(* CODESYS project TcMotion_Axis_v1.0.0.3.library
   DefaultNamespace: Tc3_Motion
   Description: Component Motion OOP Axis
   Author: victorduranm@hotmail.com
   DocFormat: reStructuredText
   Title: TcMotion_Component
   Version: 1.0.0.3
   Company: TcMotion
   Placeholder: TcMotion_Component

Project tree, tasks and I/O mapping:
  libraries: CoDeSys Library Template Interfaces, * (3S - Smart Software Solutions GmbH); Tc2_MC2, * (Beckhoff Automation GmbH); Tc2_MC2_Camming, * (Beckhoff Automation GmbH); Tc2_MC2_FlyingSaw, * (Beckhoff Automation GmbH); Tc2_Standard, * (Beckhoff Automation GmbH); Tc2_System, * (Beckhoff Automation GmbH); Tc3_DriveMotionControl, * (Beckhoff Automation GmbH); Tc3_Module, * (Beckhoff Automation GmbH)
  Component_Axis/
    function block FB_TcAxis_Codesys [ST]: AccelerationProfile, ActualPosition, ActualTorque, ActualVelocity, AxisWarning, CamIn, CombineAxes, CommunicationReady, Direction, ErrorId, GearIn, GearInPos, Halt, HaltSuperimposed, Home, HomeAbsSwitch, IsHomed, LimitSwitchNegative, LimitSwitchPositive, MotionStatus, MoveAbsolute, MoveAdditive, MoveContinuousAbsolute, MoveContinuousRelative, MoveRelative, MoveSuperimposed, MoveVelocity, PhasingAbsolute, PhasingRelative, PositionProfile, Power, PowerOn, ReadBoolParameter, ReadParameter, ReadyForPowerOn, Release, Reset, SetOverride, SetPosition, Simulation, Status, Stop, TorqueControl, VelocityProfile, WriteBoolParameter, WriteParameter
  Examples/
    program CamGearExample [ST]
    program LabelingExample [ST]
    program MAIN_Examples [ST]
    program WareHousingExample [ST]
  MsTestUnit/
    function block FB_Sum [ST]: Sum
  Project Information/
    function F_GetCompany [ST]
    function F_GetTitle [ST]
    function F_GetVersion [ST]
  TwinCAT Library Template/
    Part1Definition/
      Enums/
        data type AXIS_DIRECTION
        data type AXIS_STATUS
        data type E_AxisParameters
        data type MC_BUFFER_MODE
        data type MC_COMBINE_MODE
        data type MC_Direction
        data type MC_Error
        data type MC_ErrorID_Udint
        data type MC_ExecutionMode
        data type MC_Source
        data type MC_StartMode
        data type MC_SYNC_MODE
        data type MOTION_STATUS
      GlobalConstants/
        global variables Constants
      Interfaces/
        interface itfAxis: ActualPosition, ActualTorque, ActualVelocity, Power, ReadBoolParameter, ReadParameter, Release, Reset, SetOverride, SetPosition, WriteBoolParameter, WriteParameter, CombineAxes, GearIn, PhasingAbsolute, PhasingRelative, AccelerationProfile, Halt, HaltSuperimposed, Home, Jog, MoveAbsolute, MoveAdditive, MoveContinuousAbsolute, MoveContinuousRelative, MoveRelative, MoveSuperimposed, MoveVelocity, PositionProfile, Stop, TorqueControl, VelocityProfile, AxisWarning, CommunicationReady, Direction, Error, ErrorId, ErrorId_Udint_Status, Geared, HomeAbsSwitch, IsHomed, LimitSwitchNegative, LimitSwitchPositive, MotionStatus, PowerOn, ReadyForPowerOn, Simulation, Status
        interface itfAxis_Tc2_MC2_Camming: CamIn
        interface itfAxis_Tc2_MC2_FlyingSaw: GearInPos
        interface itfAxisCommand: update
        interface itfCamTable: Select
        interface itfCommand: Abort, Active, Busy, Command, CommandAborted, Done, Error, ErrorId, ErrorID_Udint, Wait
        interface itfContinuousAxisCommand: InVelocity
        interface itfSynchronizedAxisCommand: InSync
      Structs/
        data type MC_CAM_REF
        data type MC_COMMAND_REF
        data type ST_Command
        data type ST_MC
    VendorImplementation/
      function block TcAxis_DMC_Tc3_Direct_Motion_Control [ST]
      function block TcAxis_Tc2_MC2 [ST]: ActualPosition, ActualTorque, ActualVelocity, Power, ReadBoolParameter, ReadParameter, Release, Reset, SetOverride, SetPosition, WriteBoolParameter, WriteParameter, CombineAxes, GearIn, PhasingAbsolute, PhasingRelative, AccelerationProfile, Halt, HaltSuperimposed, Home, Jog, MoveAbsolute, MoveAdditive, MoveContinuousAbsolute, MoveContinuousRelative, MoveRelative, MoveSuperimposed, MoveVelocity, PositionProfile, Stop, TorqueControl, VelocityProfile, AxisWarning, CommunicationReady, Direction, Error, ErrorId, ErrorId_Udint_Status, Geared, HomeAbsSwitch, IsHomed, LimitSwitchNegative, LimitSwitchPositive, MotionStatus, PowerOn, ReadyForPowerOn, Simulation, Status, ACT_Cyclic_Update
      function block TcAxis_Tc2_MC2_Camming [ST]: CamIn
      function block TcAxis_Tc2_MC2_FlyingSaw [ST]: GearInPos
      function block TcAxisCommand [ST]: Abort, Active, Busy, Command, CommandAborted, Done, Error, ErrorId, ErrorID_Udint, Update, Wait
      function block TcCamTable [ST]: Select
      function block TcCommand [ST]: Abort, Active, Busy, Command, CommandAborted, Done, Error, ErrorId, ErrorID_Udint, Wait
      function block TcContinuousAxisCommand [ST]: Abort, Active, Busy, Command, CommandAborted, Done, Error, ErrorId, InVelocity, Update, Wait
      function block TcSynchronizedAxisCommand [ST]: Abort, Active, Busy, Command, CommandAborted, Done, Error, ErrorId, InSync, Update, Wait
  Version/
    global variables Global_Version
  VISUs/
*)

// TwinCAT Library Template/Part1Definition/Enums/AXIS_DIRECTION
{attribute 'qualified_only'}
{attribute 'strict'}
TYPE AXIS_DIRECTION :
(
	DirectionPositive := 0,
	DirectionNegative := 1
);
END_TYPE

// TwinCAT Library Template/Part1Definition/Enums/AXIS_STATUS
{attribute 'qualified_only'}
{attribute 'strict'}
TYPE AXIS_STATUS :
(
	ErrorStop := 0,
	Disabled := 1,
	Stopping := 2,
	Homing := 3,
	Standstill := 4,
	DiscreteMotion := 5,
	ContinuousMotion := 6,
	SynchronizedMotion := 7
);
END_TYPE

// TwinCAT Library Template/Part1Definition/Enums/E_AxisParameters
{attribute 'qualified_only'}
{attribute 'strict'}
TYPE E_AxisParameters :
(
//PLCopen specific parameters Index-Group 0x4000 + ID
    CommandedPosition := 1, //lreal taken from NcToPlc
    SWLimitForward := 2, //lreal IndexOffset= 16#0001_000E
    SWLimitBackward := 3, //lreal IndexOffset= 16#0001_000D
    EnableLimitForward := 4, //bool IndexOffset= 16#0001_000C
    EnableLimitBackward := 5, //bool IndexOffset= 16#0001_000B
    EnablePositionLagMonitoring := 6, //bool IndexOffset= 16#0002_0010
    MaxPositionLag := 7, //lreal IndexOffset= 16#0002_0012
    AxisMaxVelocity := 8, //lreal IndexOffset= 16#0000_0027
    ActualVelocity := 10, //lreal taken from NcToPlc
    CommandedVelocity := 11, //lreal taken from NcToPlc
    AxisDefaultAcceleration := 12, //lreal IndexOffset= 16#0000_0101
    AxisDefaultDeceleration := 14, //lreal IndexOffset= 16#0000_0102
    AxisDefaultJerk := 16, //lreal IndexOffset= 16#0000_0103

//Beckhoff specific parameters Index-Group 0x4000 + ID
    AxisId := 1000, //lreal IndexOffset= 16#0000_0001
    AxisManualVelocitySlow := 1001, //lreal IndexOffset= 16#0000_0008
    AxisManualVelocityFast := 1002, //lreal IndexOffset= 16#0000_0009
    AxisAccMax := 1004, //lreal IndexOffset= 16#0000_0101
    AxisDecMax := 1005, //lreal IndexOffset= 16#0000_0102
    AxisRapidTraverseVelocity := 1009, //lreal IndexOffset= 16#0000_000A
    AxisVelocityToCam := 1012, //lreal IndexOffset= 16#0000_0006
    AxisVelocityFromCam := 1013, //lreal IndexOffset= 16#0000_0007
    AxisJogIncrementForward := 1014, //lreal IndexOffset= 16#0000_0018
    AxisJogIncrementBackward := 1015, //lreal IndexOffset= 16#0000_0019
    MaxPositionLagFilterTime := 1022, //lreal IndexOffset= 16#0002_0013
    AxisEnPositionRangeMonitoring := 1023, //bool IndexOffset= 16#0000_000F
    AxisPositionRangeWindow := 1024, //lreal IndexOffset= 16#0000_0010
    AxisEnTargetPositionMonitoring:= 1025, //bool IndexOffset= 16#0000_0015
    AxisTargetPositionWindow := 1026, //lreal IndexOffset= 16#0000_0016
    AxisTargetPositionMonitoringTime := 1027, //lreal IndexOffset= 16#0000_0017
    AxisEnInTargetTimeout := 1028, //bool IndexOffset= 16#0000_0029
    AxisInTargetTimeout := 1029, //lreal IndexOffset= 16#0000_002A
    AxisEnMotionMonitoring := 1030, //bool IndexOffset= 16#0000_0011
    AxisMotionMonitoringWindow := 1031, //lreal IndexOffset= 16#0000_0028
    AxisMotionMonitoringTime := 1032, //lreal IndexOffset= 16#0000_0012
    AxisDelayTimeVeloPosition := 1033, //lreal IndexOffset= 16#0000_0104
    AxisEnLoopingDistance := 1034, //bool IndexOffset= 16#0000_0013
    AxisLoopingDistance := 1035, //lreal IndexOffset= 16#0000_0014
    AxisEnBacklashCompensation := 1036, //bool IndexOffset= 16#0000_002B
    AxisBacklash := 1037, //lreal IndexOffset= 16#0000_002C
    AxisEnDataPersistence := 1038, //bool IndexOffset= 16#0000_0030
    AxisRefVeloOnRefOutput := 1039, //lreal IndexOffset= 16#0003_0101
    AxisOverrideType := 1040, //lreal IndexOffset= 16#0000_0105
    //new since 4/2007
    AxisEncoderOffset := 1042, //lreal IndexOffset= 16#0001_0007
    AxisEncoderDirectionInverse := 1043, //bool IndexOffset= 16#0001_0008
    AxisEncoderMask := 1044, //dword IndexOffset= 16#0001_0015
    AxisEncoderModuloValue := 1045, //lreal IndexOffset= 16#0001_0009
    AxisModuloToleranceWindow := 1046, //lreal IndexOffset= 16#0001_001B
    AxisEnablePosCorrection := 1047, //bool IndexOffset= 16#0001_0016
    AxisPosCorrectionFilterTime := 1048, //lreal IndexOffset= 16#0001_0017
    //new since 1/2010
    AxisUnitInterpretation := 1049, //lreal IndexOffset= 16#0000_0026
    AxisMotorDirectionInverse := 1050, //bool  IndexOffset= 16#0003_0006
    //new since 1/2011
    AxisCycleTime := 1051, //lreal IndexOffset= 16#0000_0004
    //new since 5/2011
    AxisFastStopSignalType := 1052, //dword IndexOffset= 16#0000_001E
    AxisFastAcc := 1053, //lreal IndexOffset= 16#0000_010A
    AxisFastDec := 1054, //lreal IndexOffset= 16#0000_010B
    AxisFastJerk := 1055, //lreal IndexOffset= 16#0000_010C
    // new since 1/2012 *)
    AxisEncoderScalingNumerator := 1056, //lreal IndexOffset= 16#0001_0023 - available in Tc3
    AxisEncoderScalingDenominator := 1057, //lreal IndexOffset= 16#0001_0024 - available in Tc3
    (* new since 7/2016 *)
    AxisVeloJumpFactor := 1060, //lreal IndexOffset= 16#0000_0106
    AxisToleranceBallAuxAxis := 1061, //lreal IndexOffset= 16#0000_0108
    AxisMaxPositionDeviationAuxAxis := 1062, //lreal IndexOffset= 16#0000_0109
    AxisErrorPropagationMode := 1063, //dword IndexOffset= 16#0000_001A
    AxisErrorPropagationDelay := 1064, //lreal IndexOffset= 16#0000_001B
    AxisCoupleSlaveToActualValues := 1065, //bool IndexOffset= 16#0000_001C
    AxisAllowMotionCmdToSlaveAxis := 1066, //bool IndexOffset= 16#0000_0020
    AxisAllowMotionCmdToExtSetAxis := 1067, //bool IndexOffset= 16#0000_0021
    AxisEncoderSubMask := 1068, //dword IndexOffset= 16#0001_0108
    AxisEncoderReferenceSystem := 1069, //dword IndexOffset= 16#0001_0019
    AxisEncoderPositionFilterPT1 := 1070, //lreal IndexOffset= 16#0001_0010
    AxisEncoderVelocityFilterPT1 := 1071, //lreal IndexOffset= 16#0001_0011
    AxisEncoderAccelerationFilterPT1 := 1072, //lreal IndexOffset= 16#0001_0012
    AxisEncoderMode := 1073, //dword IndexOffset= 16#0001_000A
    AxisEncoderHomingInvDirCamSearch := 1074, //bool IndexOffset= 16#0001_0101
    AxisEncoderHomingInvDirSyncSearch := 1075, //bool IndexOffset= 16#0001_0102
    AxisEncoderHomingCalibValue := 1076, //lreal IndexOffset= 16#0001_0103
    AxisEncoderReferenceMode := 1077, //dword IndexOffset= 16#0001_0107
    AxisRefVeloOutputRatio := 1078, //lreal IndexOffset= 16#0003_0102
    AxisDrivePositionOutputScaling := 1079, //lreal IndexOffset= 16#0003_0109
    AxisDriveVelocityOutputScaling := 1080, //lreal IndexOffset= 16#0003_0105
    AxisDriveVelocityOutputDelay := 1081, //lreal IndexOffset= 16#0003_010D
    AxisDriveMinOutputLimitation := 1082, //lreal IndexOffset= 16#0003_000B
    AxisDriveMaxOutputLimitation := 1083, //lreal IndexOffset= 16#0003_000C
    AxisTorqueInputScaling := 1084, //lreal IndexOffset= 16#0003_0031 - available in Tc3
    AxisTorqueInputFilterPT1 := 1085, //lreal IndexOffset= 16#0003_0032 - available in Tc3
    AxisTorqueDerivationInputFilterPT1 := 1086, //lreal IndexOffset= 16#0003_0033 - available in Tc3
    AxisTorqueOutputScaling := 1087, //lreal IndexOffset= 16#0003_010B
    AxisTorqueOutputDelay := 1088, //lreal IndexOffset= 16#0003_010F
    AxisAccelerationOutputScaling := 1089, //lreal IndexOffset= 16#0003_010A
    AxisAccelerationOutputDelay := 1090, //lreal IndexOffset= 16#0003_010E
    AxisDrivePositionOutputSmoothFilterType := 1091, //dword IndexOffset= 16#0003_0110
    AxisDrivePositionOutputSmoothFilterTime := 1092, //lreal IndexOffset= 16#0003_0111
    AxisDrivePositionOutputSmoothFilterOrder := 1093, //dword IndexOffset= 16#0003_0112
    AxisDriveMode := 1094, //dword IndexOffset= 16#0003_000A
    AxisDriftCompensationOffset := 1095, //lreal IndexOffset= 16#0003_0104
    AxisPositionControlKv := 1096, //lreal IndexOffset= 16#0002_0102
    AxisCtrlVelocityPreCtrlWeight := 1097, //lreal IndexOffset= 16#0002_000B
    AxisControllerMode := 1098, //dword IndexOffset= 16#0002_000A
    AxisCtrlAutoOffset := 1099, //bool IndexOffset= 16#0002_0110
    AxisCtrlAutoOffsetTimer := 1100, //lreal IndexOffset= 16#0002_0115
    AxisCtrlAutoOffsetLimit := 1101, //lreal IndexOffset= 16#0002_0114
    AxisSlaveCouplingControlKcp := 1102, //lreal IndexOffset= 16#0002_010F
    AxisCtrlOutputLimit := 1103, //lreal IndexOffset= 16#0002_0100

//Beckhoff specific axis status information - READ ONLY Index-Group 0x4100 + ID
    AxisTargetPosition := 2000, //lreal IndexOffset= 16#0000_0013
    AxisRemainingTimeToGo := 2001, //lreal IndexOffset= 16#0000_0014
    AxisRemainingDistanceToGo := 2002, //lreal IndexOffset= 16#0000_0022, 16#0000_0042

//Beckhoff specific axis functions
    //read/write gear ratio of a slave
    AxisGearRatio := 3000, //lreal read: IndexGroup=0x4100+ID, IdxOffset=16#0000_0022,
                                 //write:IndexGroup=0x4200+ID, IdxOffset=16#0000_0042

//Beckhoff specific other parameters
    //new since 1/2011
    NcSafCycleTime := 4000, //lreal IndexOffset= 16#0000_0010
    NcSvbCycleTime := 4001 //lreal IndexOffset= 16#0000_0012

);
END_TYPE

// TwinCAT Library Template/Part1Definition/Enums/MC_BUFFER_MODE
{attribute 'qualified_only'}
{attribute 'strict'}
TYPE MC_BUFFER_MODE :
(
	mcAborting := 0,
	mcBuffered := 1,
	mcBlendingLow := 2,
	mcBlendingPrevious := 3,
	mcBlendingNext := 4,
	mcBlendingHigh := 5
);
END_TYPE

// TwinCAT Library Template/Part1Definition/Enums/MC_COMBINE_MODE
{attribute 'qualified_only'}
{attribute 'strict'}
TYPE MC_COMBINE_MODE :
(
	enum_member := 0
);
END_TYPE

// TwinCAT Library Template/Part1Definition/Enums/MC_Direction
{attribute 'qualified_only'}
{attribute 'strict'}
TYPE MC_Direction :
(
	mcPositiveDirection := 0,
	mcShortestWay := 1,
	mcNegativeDirection := 2,
	mcCurrentDirection := 3
);
END_TYPE

// TwinCAT Library Template/Part1Definition/Enums/MC_Error
{attribute 'qualified_only'}
//{attribute 'conditionalshow' := 'SomeText'}
//{attribute 'conditionalshow'}
//{attribute 'hide'}
TYPE MC_Error : (NO_ERROR, TIME_OUT); END_TYPE

// TwinCAT Library Template/Part1Definition/Enums/MC_ErrorID_Udint
TYPE MC_ErrorID_Udint : UDINT; END_TYPE

// TwinCAT Library Template/Part1Definition/Enums/MC_ExecutionMode
{attribute 'qualified_only'}
{attribute 'strict'}
TYPE MC_ExecutionMode :
(
	mcImmediatly := 0,
	mcQueue := 1
);
END_TYPE

// TwinCAT Library Template/Part1Definition/Enums/MC_Source
{attribute 'qualified_only'}
{attribute 'strict'}
TYPE MC_Source :
(
	mcSetValue := 0,
	mcActualValue := 1
);
END_TYPE

// TwinCAT Library Template/Part1Definition/Enums/MC_StartMode
{attribute 'qualified_only'}
{attribute 'strict'}
TYPE MC_StartMode :
(
	mcAbsolute := 0,
	mcRelative := 1,
	mcRampIn := 2
);
END_TYPE

// TwinCAT Library Template/Part1Definition/Enums/MC_SYNC_MODE
{attribute 'qualified_only'}
{attribute 'strict'}
TYPE MC_SYNC_MODE :
(
	enum_member := 0
);
END_TYPE

// TwinCAT Library Template/Part1Definition/Enums/MOTION_STATUS
{attribute 'qualified_only'}
{attribute 'strict'}
TYPE MOTION_STATUS :
(
	ConstantVelocity := 0,
	Accelerating := 1,
	Decelerating :=2
);
END_TYPE

// TwinCAT Library Template/Part1Definition/Structs/MC_CAM_REF
TYPE MC_CAM_REF :
STRUCT
END_STRUCT
END_TYPE

// TwinCAT Library Template/Part1Definition/Structs/MC_COMMAND_REF
TYPE MC_COMMAND_REF :
STRUCT
	CommandId: INT;
END_STRUCT
END_TYPE

// TwinCAT Library Template/Part1Definition/Structs/ST_Command
TYPE ST_Command :
STRUCT
	Active 			: BOOL;
	Busy 			: BOOL;
	Command 		: MC_COMMAND_REF;
	CommandAborted 	: BOOL;
	Done           	: BOOL;
	Error    		: BOOL;
	ErrorId        	: MC_Error;
	ErrorID_Udint	: MC_ErrorID_Udint;
END_STRUCT
END_TYPE

// TwinCAT Library Template/Part1Definition/Structs/ST_MC
TYPE ST_MC :
STRUCT
	Power 			: Tc2_MC2.MC_POWER;
	MoveAbsolute 	: Tc2_MC2.MC_MoveAbsolute;	
	MoveRelative 	: Tc2_MC2.MC_MoveRelative;
END_STRUCT
END_TYPE

// TwinCAT Library Template/Part1Definition/GlobalConstants/Constants
//{attribute 'conditionalshow' := 'SomeText'}
//{attribute 'conditionalshow'}
//{attribute 'hide'}
VAR_GLOBAL CONSTANT
END_VAR

// Version/Global_Version
{attribute 'TcGenerated'}
{attribute 'no-analysis'}
{attribute 'linkalways'}
// This function has been automatically generated from the project information.
VAR_GLOBAL CONSTANT
	{attribute 'const_non_replaced'}
	stLibVersion_TcMotion_Component : ST_LibVersion := (iMajor := 1, iMinor := 0, iBuild := 0, iRevision := 3, nFlags := 0, sVersion := '1.0.0.3');
END_VAR

// Component_Axis/FB_TcAxis_Codesys
FUNCTION_BLOCK FB_TcAxis_Codesys IMPLEMENTS TMP.itfAxis
VAR_INPUT
END_VAR
VAR_OUTPUT
END_VAR
VAR
END_VAR

{warning 'Agregar implementación de método'}
METHOD AccelerationProfile : itfCommand
VAR_INPUT
	TimeScale	: REAL;
	AccelerationScale	: REAL;
	Offset	: REAL;
	BufferMode	: MC_BUFFER_MODE;
END_VAR
// NETWORK 1
END_METHOD

{warning 'Agregar implementación de propiedad'}
PROPERTY ActualPosition : REAL
GET
// NETWORK 1
END_GET
END_PROPERTY

{warning 'Agregar implementación de propiedad'}
PROPERTY ActualTorque : REAL
GET
// NETWORK 1
END_GET
END_PROPERTY

{warning 'Agregar implementación de propiedad'}
PROPERTY ActualVelocity : REAL
GET
// NETWORK 1
END_GET
END_PROPERTY

{warning 'Agregar implementación de propiedad'}
PROPERTY AxisWarning : BOOL
GET
// NETWORK 1
END_GET
END_PROPERTY

{warning 'Agregar implementación de método'}
METHOD CamIn : itfSynchronizedAxisCommand
VAR_INPUT
	Master	: itfAxis;
	MasterOffset	: REAL;
	SlaveOffset	: REAL;
	MasterScaling	: REAL;
	SlaveScaling	: REAL;
	MasterStartDistance	: REAL;
	MasterSyncPosition	: REAL;
	StartMode	: MC_StartMode;
	MasterValueSource	: MC_Source;
	CamTable	: itfCamTable;
	BufferMode	: MC_BUFFER_MODE;
END_VAR
// NETWORK 1
END_METHOD

{warning 'Agregar implementación de método'}
METHOD CombineAxes : itfSynchronizedAxisCommand
VAR_INPUT
	Master1	: itfAxis;
	Master2	: itfAxis;
	CombineMode	: MC_COMBINE_MODE;
	GearRatioNumeratorM1	: INT;
	GearRatioDenominatorM1	: INT;
	GearRatioNumeratorM2	: INT;
	GearRatioDenominatorM2	: INT;
	MasterValueSourceM1	: MC_SOURCE;
	MasterValueSourceM2	: MC_SOURCE;
	BufferMode	: MC_BUFFER_MODE;
END_VAR
// NETWORK 1
END_METHOD

{warning 'Agregar implementación de propiedad'}
PROPERTY CommunicationReady : BOOL
GET
// NETWORK 1
END_GET
END_PROPERTY

{warning 'Agregar implementación de propiedad'}
PROPERTY Direction : AXIS_DIRECTION
GET
// NETWORK 1
END_GET
END_PROPERTY

{warning 'Agregar implementación de propiedad'}
PROPERTY ErrorId : WORD
GET
// NETWORK 1
END_GET
END_PROPERTY

{warning 'Agregar implementación de método'}
METHOD GearIn : itfSynchronizedAxisCommand
VAR_INPUT
	Master	: itfAxis;
	Ratio	: REAL;
	MasterValueSource	: INT;
	Acceleration	: REAL;
	Deceleration	: REAL;
	Jerk	: REAL;
	BufferMode	: MC_BUFFER_MODE;
END_VAR
// NETWORK 1
END_METHOD

{warning 'Agregar implementación de método'}
METHOD GearInPos : itfSynchronizedAxisCommand
VAR_INPUT
	Master	: itfAxis;
	RatioNumerator	: REAL;
	RatioDenominator	: REAL;
	MasterValueSource	: MC_SOURCE;
	MasterSyncPosition	: REAL;
	SlaveSyncPosition	: REAL;
	SyncMode	: MC_SYNC_MODE;
	MasterStartDistance	: REAL;
	Velocity	: REAL;
	Acceleration	: REAL;
	Deceleration	: REAL;
	Jerk	: REAL;
	BufferMode	: MC_BUFFER_MODE;
END_VAR
// NETWORK 1
END_METHOD

{warning 'Agregar implementación de método'}
METHOD Halt : itfAxisCommand
VAR_INPUT
	Deceleration	: REAL;
	Jerk	: REAL;
	BufferMode	: MC_BUFFER_MODE;
END_VAR
// NETWORK 1
END_METHOD

{warning 'Agregar implementación de método'}
METHOD HaltSuperimposed : itfAxisCommand
VAR_INPUT
	Deceleration	: REAL;
	Jerk	: REAL;
END_VAR
// NETWORK 1
END_METHOD

{warning 'Agregar implementación de método'}
METHOD Home : itfAxisCommand
VAR_INPUT
	Position	: REAL;
	Velocity	: REAL;
	EndVelocity	: REAL;
	Acceleration	: REAL;
	Deceleration	: REAL;
	Jerk	: REAL;
	Direction	: MC_Direction;
	HomingMode	: INT;
	BufferMode	: MC_BUFFER_MODE;
END_VAR
// NETWORK 1
END_METHOD

{warning 'Agregar implementación de propiedad'}
PROPERTY HomeAbsSwitch : BOOL
GET
// NETWORK 1
END_GET
END_PROPERTY

{warning 'Agregar implementación de propiedad'}
PROPERTY IsHomed : BOOL
GET
// NETWORK 1
END_GET
END_PROPERTY

{warning 'Agregar implementación de propiedad'}
PROPERTY LimitSwitchNegative : BOOL
GET
// NETWORK 1
END_GET
END_PROPERTY

{warning 'Agregar implementación de propiedad'}
PROPERTY LimitSwitchPositive : BOOL
GET
// NETWORK 1
END_GET
END_PROPERTY

{warning 'Agregar implementación de propiedad'}
PROPERTY MotionStatus : MOTION_STATUS
GET
// NETWORK 1
END_GET
END_PROPERTY

{warning 'Agregar implementación de método'}
METHOD MoveAbsolute : itfAxisCommand
VAR_INPUT
	Position	: REAL;
	Velocity	: REAL;
	Acceleration	: REAL;
	Deceleration	: REAL;
	Jerk	: REAL;
	Direction	: MC_Direction;
	BufferMode	: MC_BUFFER_MODE;
END_VAR
// NETWORK 1
END_METHOD

{warning 'Agregar implementación de método'}
METHOD MoveAdditive : itfAxisCommand
VAR_INPUT
	Distance	: REAL;
	Velocity	: REAL;
	Acceleration	: REAL;
	Deceleration	: REAL;
	Jerk	: REAL;
	BufferMode	: MC_BUFFER_MODE;
END_VAR
// NETWORK 1
END_METHOD

{warning 'Agregar implementación de método'}
METHOD MoveContinuousAbsolute : itfContinuousAxisCommand
VAR_INPUT
	Position	: REAL;
	EndVelocity	: REAL;
	Velocity	: REAL;
	Acceleration	: REAL;
	Deceleration	: REAL;
	Jerk	: REAL;
	Direction	: MC_DIRECTION;
	BufferMode	: MC_BUFFER_MODE;
END_VAR
// NETWORK 1
END_METHOD

{warning 'Agregar implementación de método'}
METHOD MoveContinuousRelative : itfContinuousAxisCommand
VAR_INPUT
	Distance	: REAL;
	EndVelocity	: REAL;
	Velocity	: REAL;
	Acceleration	: REAL;
	Deceleration	: REAL;
	Jerk	: REAL;
	Direction	: MC_DIRECTION;
	BufferMode	: MC_BUFFER_MODE;
END_VAR
// NETWORK 1
END_METHOD

{warning 'Agregar implementación de método'}
METHOD MoveRelative : itfAxisCommand
VAR_INPUT
	Distance	: REAL;
	Velocity	: REAL;
	Acceleration	: REAL;
	Deceleration	: REAL;
	Jerk	: REAL;
	BufferMode	: MC_BUFFER_MODE;
END_VAR
// NETWORK 1
END_METHOD

{warning 'Agregar implementación de método'}
METHOD MoveSuperimposed : itfAxisCommand
VAR_INPUT
	Distance	: REAL;
	VelocityDiff	: REAL;
	Acceleration	: REAL;
	Deceleration	: REAL;
	Jerk	: REAL;
END_VAR
// NETWORK 1
END_METHOD

{warning 'Agregar implementación de método'}
METHOD MoveVelocity : itfContinuousAxisCommand
VAR_INPUT
	Velocity	: REAL;
	Acceleration	: REAL;
	Deceleration	: REAL;
	Jerk	: REAL;
	Direction	: MC_Direction;
	BufferMode	: MC_BUFFER_MODE;
END_VAR
// NETWORK 1
END_METHOD

{warning 'Agregar implementación de método'}
METHOD PhasingAbsolute : itfSynchronizedAxisCommand
VAR_INPUT
	Master	: itfAxis;
	PhaseShift	: REAL;
	Velocity	: REAL;
	Acceleration	: REAL;
	Deceleration	: REAL;
	Jerk	: REAL;
	BufferMode	: MC_BUFFER_MODE;
END_VAR
// NETWORK 1
END_METHOD

{warning 'Agregar implementación de método'}
METHOD PhasingRelative : itfSynchronizedAxisCommand
VAR_INPUT
	Master	: itfAxis;
	PhaseShift	: REAL;
	Velocity	: REAL;
	Acceleration	: REAL;
	Deceleration	: REAL;
	Jerk	: REAL;
	BufferMode	: MC_BUFFER_MODE;
END_VAR
// NETWORK 1
END_METHOD

{warning 'Agregar implementación de método'}
METHOD PositionProfile : itfCommand
VAR_INPUT
	TimeScale	: REAL;
	PositionScale	: REAL;
	Offset	: REAL;
	BufferMode	: MC_BUFFER_MODE;
END_VAR
// NETWORK 1
END_METHOD

{warning 'Agregar implementación de método'}
METHOD Power : itfCommand
VAR_INPUT
	Enable	: BOOL;
	EnablePositive	: BOOL;
	EnableNegative	: BOOL;
END_VAR
// NETWORK 1
END_METHOD

{warning 'Agregar implementación de propiedad'}
PROPERTY PowerOn : BOOL
GET
// NETWORK 1
END_GET
END_PROPERTY

{warning 'Agregar implementación de método'}
METHOD ReadBoolParameter : MC_Error
VAR_INPUT
	ParameterNumber	: INT;
END_VAR
VAR_OUTPUT
	Value	: BOOL;
END_VAR
// NETWORK 1
END_METHOD

{warning 'Agregar implementación de método'}
METHOD ReadParameter : MC_Error
VAR_INPUT
	ParameterNumber	: INT;
END_VAR
VAR_OUTPUT
	Value	: REAL;
END_VAR
// NETWORK 1
END_METHOD

{warning 'Agregar implementación de propiedad'}
PROPERTY ReadyForPowerOn : BOOL
GET
// NETWORK 1
END_GET
END_PROPERTY

{warning 'Agregar implementación de método'}
METHOD Release : MC_Error
// NETWORK 1
END_METHOD

{warning 'Agregar implementación de método'}
METHOD Reset : itfCommand
// NETWORK 1
END_METHOD

{warning 'Agregar implementación de método'}
METHOD SetOverride : MC_Error
VAR_INPUT
	VelFactor	: REAL;
	AccFactor	: REAL;
	JerkFactor	: REAL;
END_VAR
// NETWORK 1
END_METHOD

{warning 'Agregar implementación de método'}
METHOD SetPosition : itfCommand
VAR_INPUT
	Position	: REAL;
	Relative	: BOOL;
	ExecutionMode	: MC_ExecutionMode;
END_VAR
// NETWORK 1
END_METHOD

{warning 'Agregar implementación de propiedad'}
PROPERTY Simulation : BOOL
GET
// NETWORK 1
END_GET
END_PROPERTY

{warning 'Agregar implementación de propiedad'}
PROPERTY Status : AXIS_STATUS
GET
// NETWORK 1
END_GET
END_PROPERTY

{warning 'Agregar implementación de método'}
METHOD Stop : itfAxisCommand
VAR_INPUT
	Deceleration	: REAL;
	Jerk	: REAL;
END_VAR
// NETWORK 1
END_METHOD

{warning 'Agregar implementación de método'}
METHOD TorqueControl : itfAxisCommand
VAR_INPUT
	Torque	: REAL;
	TorqueRamp	: REAL;
	Velocity	: REAL;
	Acceleration	: REAL;
	Deceleration	: REAL;
	Jerk	: REAL;
	Direction	: MC_DIRECTION;
	BufferMode	: MC_BUFFER_MODE;
END_VAR
// NETWORK 1
END_METHOD

{warning 'Agregar implementación de método'}
METHOD VelocityProfile : itfCommand
VAR_INPUT
	TimeScale	: REAL;
	VelocityScale	: REAL;
	Offset	: REAL;
	BufferMode	: MC_BUFFER_MODE;
END_VAR
// NETWORK 1
END_METHOD

{warning 'Agregar implementación de método'}
METHOD WriteBoolParameter : MC_Error
VAR_INPUT
	ParameterNumber	: INT;
	Value	: BOOL;
END_VAR
// NETWORK 1
END_METHOD

{warning 'Agregar implementación de método'}
METHOD WriteParameter : MC_Error
VAR_INPUT
	ParameterNumber	: INT;
	Value	: REAL;
END_VAR
// NETWORK 1
END_METHOD

END_FUNCTION_BLOCK

// TwinCAT Library Template/Part1Definition/Interfaces/itfAxis
INTERFACE itfAxis

{warning 'add property implementation'}
PROPERTY ActualPosition : REAL
GET
END_GET
END_PROPERTY

{warning 'add property implementation'}
PROPERTY ActualTorque : REAL
GET
END_GET
END_PROPERTY

{warning 'add property implementation'}
PROPERTY ActualVelocity : REAL
GET
END_GET
END_PROPERTY

{attribute 'TcRpcEnable'}
METHOD Power 		: itfCommand
VAR_INPUT
	Enable			: BOOL;
	EnablePositive	: BOOL;
	EnableNegative	: BOOL;
END_VAR
END_METHOD

{warning 'add method implementation '}
METHOD ReadBoolParameter 	: MC_Error
VAR_INPUT
	ParameterNumber			: INT;
END_VAR
VAR_OUTPUT
	Value					: BOOL;
END_VAR
END_METHOD

{warning 'add method implementation '}
METHOD ReadParameter 	: MC_Error
VAR_INPUT
	ParameterNumber		: INT;
END_VAR
VAR_OUTPUT
	Value				: REAL;
END_VAR
END_METHOD

{warning 'add method implementation '}
METHOD Release : MC_Error
END_METHOD

{attribute 'TcRpcEnable'}
METHOD Reset : itfCommand
END_METHOD

{warning 'add method implementation '}
METHOD SetOverride 	: MC_Error
VAR_INPUT
	VelFactor		: REAL;
	AccFactor		: REAL;
	JerkFactor		: REAL;
END_VAR
END_METHOD

{warning 'add method implementation '}
METHOD SetPosition 	: itfCommand
VAR_INPUT
	Position		: REAL;
	Relative		: BOOL;
//	ExecutionMode	: MC_ExecutionMode;
	ExecutionMode	: Tc2_MC2.ST_SetPositionOptions;
END_VAR
END_METHOD

{warning 'add method implementation '}
METHOD WriteBoolParameter 	: MC_Error
VAR_INPUT
	ParameterNumber			: INT;
	Value					: BOOL;
END_VAR
END_METHOD

{warning 'add method implementation '}
METHOD WriteParameter 	: MC_Error
VAR_INPUT
	ParameterNumber		: INT;
	Value				: REAL;
END_VAR
END_METHOD

{warning 'add method implementation '}
METHOD CombineAxes 			: itfSynchronizedAxisCommand
VAR_INPUT
	Master1					: itfAxis;
	Master2					: itfAxis;
	CombineMode				: MC_COMBINE_MODE;
	GearRatioNumeratorM1	: INT;
	GearRatioDenominatorM1	: INT;
	GearRatioNumeratorM2	: INT;
	GearRatioDenominatorM2	: INT;
	MasterValueSourceM1		: MC_SOURCE;
	MasterValueSourceM2		: MC_SOURCE;
	BufferMode				: MC_BUFFER_MODE;
END_VAR
END_METHOD

{attribute 'TcRpcEnable'}
METHOD GearIn 			: itfSynchronizedAxisCommand
VAR_INPUT
//	Master				: itfAxis;
//	Master				: Tc2_MC2.AXIS_REF;
//	Slave				: Tc2_MC2.AXIS_REF;		
//	Ratio				: REAL;
//	MasterValueSource	: INT;
	RatioNumerator		: LREAL;
	RatioDenominator	: UINT;
	Acceleration		: REAL;
	Deceleration		: REAL;
	Jerk				: REAL;
	BufferMode			: MC_BUFFER_MODE;
//	BufferMode			: Tc2_MC2.MC_BufferMode;
//	Options             : Tc2_MC2.ST_GearInOptions;
END_VAR

VAR_IN_OUT 
	Slave				: Tc2_MC2.AXIS_REF;	
END_VAR
END_METHOD

{warning 'add method implementation '}
METHOD PhasingAbsolute 	: itfSynchronizedAxisCommand
VAR_INPUT
//	Master				: itfAxis;
	Master				: Tc2_MC2.AXIS_REF;
	Slave				: Tc2_MC2.AXIS_REF;		
	PhaseShift			: REAL;
	Velocity			: REAL;
	Acceleration		: REAL;
	Deceleration		: REAL;
	Jerk				: REAL;
	BufferMode			: MC_BUFFER_MODE;
END_VAR
END_METHOD

{warning 'add method implementation '}
METHOD PhasingRelative 	: itfSynchronizedAxisCommand
VAR_INPUT
//	Master				: itfAxis;
	Master				: Tc2_MC2.AXIS_REF;
	Slave				: Tc2_MC2.AXIS_REF;		
	PhaseShift			: REAL;
	Velocity			: REAL;
	Acceleration		: REAL;
	Deceleration		: REAL;
	Jerk				: REAL;
	BufferMode			: MC_BUFFER_MODE;
END_VAR
END_METHOD

{warning 'add method implementation '}
METHOD AccelerationProfile 	: itfCommand
VAR_INPUT
	TimeScale				: REAL;
	AccelerationScale		: REAL;
	Offset					: REAL;
	BufferMode				: MC_BUFFER_MODE;
END_VAR
END_METHOD

{warning 'add method implementation '}
METHOD Halt 		: itfAxisCommand
VAR_INPUT
	Deceleration	: REAL;
	Jerk			: REAL;
	BufferMode		: MC_BUFFER_MODE;
END_VAR
END_METHOD

{warning 'add method implementation '}
METHOD HaltSuperimposed : itfAxisCommand
VAR_INPUT
	Deceleration		: REAL;
	Jerk				: REAL;
END_VAR
END_METHOD

{warning 'add method implementation '}
METHOD Home 		: itfAxisCommand
VAR_INPUT
	Position		: REAL;
	Velocity		: REAL;
	EndVelocity		: REAL;
	Acceleration	: REAL;
	Deceleration	: REAL;
	Jerk			: REAL;
	Direction		: MC_Direction;
	HomingMode		: INT;
	BufferMode		: MC_BUFFER_MODE;
END_VAR
END_METHOD

{warning 'add method implementation '}
METHOD Jog 			: itfAxisCommand
VAR_INPUT
    JogForward 		: BOOL;
    JogBackwards 	: BOOL;
    Mode     		: Tc2_MC2.E_JogMode;
    Position        : LREAL;
    Velocity        : LREAL;
    Acceleration 	: LREAL;
    Deceleration 	: LREAL;
    Jerk     		: LREAL;
END_VAR
END_METHOD

{attribute 'TcRpcEnable'}
METHOD MoveAbsolute : itfAxisCommand
VAR_INPUT
	Position		: REAL;
	Velocity		: REAL;
	Acceleration	: REAL;
	Deceleration	: REAL;
	Jerk			: REAL;
	Direction		: MC_Direction;
	BufferMode		: MC_BUFFER_MODE;
END_VAR
END_METHOD

{warning 'add method implementation '}
METHOD MoveAdditive : itfAxisCommand
VAR_INPUT
	Distance		: REAL;
	Velocity		: REAL;
	Acceleration	: REAL;
	Deceleration	: REAL;
	Jerk			: REAL;
	BufferMode		: MC_BUFFER_MODE;
END_VAR
END_METHOD

{warning 'add method implementation '}
METHOD MoveContinuousAbsolute 	: itfContinuousAxisCommand
VAR_INPUT
	Position					: REAL;
	EndVelocity					: REAL;
	Velocity					: REAL;
	Acceleration				: REAL;
	Deceleration				: REAL;
	Jerk						: REAL;
	Direction					: MC_DIRECTION;
	BufferMode					: MC_BUFFER_MODE;
END_VAR
END_METHOD

{warning 'add method implementation '}
METHOD MoveContinuousRelative 	: itfContinuousAxisCommand
VAR_INPUT
	Distance					: REAL;
	EndVelocity					: REAL;
	Velocity					: REAL;
	Acceleration				: REAL;
	Deceleration				: REAL;
	Jerk						: REAL;
	Direction					: MC_DIRECTION;
	BufferMode					: MC_BUFFER_MODE;
END_VAR
END_METHOD

{attribute 'TcRpcEnable'}
METHOD MoveRelative : itfAxisCommand
VAR_INPUT
	Distance		: REAL;
	Velocity		: REAL;
	Acceleration	: REAL;
	Deceleration	: REAL;
	Jerk			: REAL;
	BufferMode		: MC_BUFFER_MODE;
END_VAR
END_METHOD

{warning 'add method implementation '}
METHOD MoveSuperimposed : itfAxisCommand
VAR_INPUT
	Distance			: REAL;
	VelocityDiff		: REAL;
	Acceleration		: REAL;
	Deceleration		: REAL;
	Jerk				: REAL;
END_VAR
END_METHOD

{warning 'add method implementation '}
METHOD MoveVelocity : itfContinuousAxisCommand
VAR_INPUT
	Velocity		: REAL;
	Acceleration	: REAL;
	Deceleration	: REAL;
	Jerk			: REAL;
	Direction		: MC_Direction;
	BufferMode		: MC_BUFFER_MODE;
END_VAR
END_METHOD

{warning 'add method implementation '}
METHOD PositionProfile : itfCommand
VAR_INPUT
	TimeScale			: REAL;
	PositionScale		: REAL;
	Offset				: REAL;
	BufferMode			: MC_BUFFER_MODE;
END_VAR
END_METHOD

{warning 'add method implementation '}
METHOD Stop 		: itfAxisCommand
VAR_INPUT
	Deceleration	: REAL;
	Jerk			: REAL;
END_VAR
END_METHOD

{warning 'add method implementation '}
METHOD TorqueControl	: itfAxisCommand
VAR_INPUT
	Torque				: REAL;
	TorqueRamp			: REAL;
	Velocity			: REAL;
	Acceleration		: REAL;
	Deceleration		: REAL;
	Jerk				: REAL;
	Direction			: MC_DIRECTION;
	BufferMode			: MC_BUFFER_MODE;
END_VAR
END_METHOD

{warning 'add method implementation '}
METHOD VelocityProfile 	: itfCommand
VAR_INPUT
	TimeScale			: REAL;
	VelocityScale		: REAL;
	Offset				: REAL;
	BufferMode			: MC_BUFFER_MODE;
END_VAR
END_METHOD

{warning 'add property implementation'}
PROPERTY AxisWarning : BOOL
GET
END_GET
END_PROPERTY

{warning 'add property implementation'}
PROPERTY CommunicationReady : BOOL
GET
END_GET
END_PROPERTY

{warning 'add property implementation'}
PROPERTY Direction : AXIS_DIRECTION
GET
END_GET
END_PROPERTY

PROPERTY Error : BOOL
GET
END_GET
END_PROPERTY

{warning 'add property implementation'}
PROPERTY ErrorId : WORD
GET
END_GET
END_PROPERTY

PROPERTY ErrorId_Udint_Status : UDINT
GET
END_GET
END_PROPERTY

PROPERTY Geared : BOOL
GET
END_GET
END_PROPERTY

{warning 'add property implementation'}
PROPERTY HomeAbsSwitch : BOOL
GET
END_GET
END_PROPERTY


PROPERTY IsHomed : BOOL
GET
END_GET
END_PROPERTY

{warning 'add property implementation'}
PROPERTY LimitSwitchNegative : BOOL
GET
END_GET
END_PROPERTY

{warning 'add property implementation'}
PROPERTY LimitSwitchPositive : BOOL
GET
END_GET
END_PROPERTY

{warning 'add property implementation'}
PROPERTY MotionStatus : MOTION_STATUS
GET
END_GET
END_PROPERTY

{attribute ‘monitoring’ := ‘call’}
PROPERTY PowerOn : BOOL
GET
END_GET
END_PROPERTY

{warning 'add property implementation'}
PROPERTY ReadyForPowerOn : BOOL
GET
END_GET
END_PROPERTY

{warning 'add property implementation'}
PROPERTY Simulation : BOOL
GET
END_GET
END_PROPERTY

{attribute ‘monitoring’ := ‘call’}
PROPERTY Status : Tc2_MC2.MC_AxisStates
GET
END_GET
END_PROPERTY

END_INTERFACE

// TwinCAT Library Template/Part1Definition/Interfaces/itfCommand
INTERFACE itfCommand

METHOD Abort : MC_Error
VAR_INPUT
END_VAR
END_METHOD

PROPERTY Active : BOOL
GET
END_GET
SET
END_SET
END_PROPERTY

PROPERTY Busy : BOOL
GET
END_GET
SET
END_SET
END_PROPERTY

PROPERTY Command : MC_COMMAND_REF
GET
END_GET
SET
END_SET
END_PROPERTY

PROPERTY CommandAborted : BOOL
GET
END_GET
SET
END_SET
END_PROPERTY

PROPERTY Done : BOOL
GET
END_GET
SET
END_SET
END_PROPERTY

PROPERTY Error : BOOL
GET
END_GET
SET
END_SET
END_PROPERTY

PROPERTY ErrorId : MC_Error
GET
END_GET
SET
END_SET
END_PROPERTY

PROPERTY ErrorID_Udint : MC_ErrorID_Udint
GET
END_GET
SET
END_SET
END_PROPERTY

METHOD Wait 		: MC_Error // This method only makes sense in the IEC 61499 environment
VAR_INPUT
	Timeout		 	: TIME;
	AbortOnTimeout 	: BOOL; 
END_VAR
END_METHOD

END_INTERFACE

// TwinCAT Library Template/Part1Definition/Interfaces/itfSynchronizedAxisCommand
INTERFACE itfSynchronizedAxisCommand EXTENDS itfAxisCommand

PROPERTY InSync : BOOL
GET
END_GET
END_PROPERTY

END_INTERFACE

// TwinCAT Library Template/Part1Definition/Interfaces/itfAxisCommand
INTERFACE itfAxisCommand EXTENDS itfCommand

METHOD Update 		: MC_Error
VAR_INPUT
	Position 		: REAL;
	Velocity 		: REAL;
	EndVelocity 	: REAL;
	Acceleration 	: REAL;
	Deceleration 	: REAL;
	Jerk 			: REAL;
END_VAR
END_METHOD

END_INTERFACE

// TwinCAT Library Template/Part1Definition/Interfaces/itfContinuousAxisCommand
INTERFACE itfContinuousAxisCommand EXTENDS itfAxisCommand

PROPERTY InVelocity : BOOL
GET
END_GET
END_PROPERTY

END_INTERFACE

// TwinCAT Library Template/Part1Definition/Interfaces/itfCamTable
INTERFACE itfCamTable

METHOD Select		: itfCommand
VAR_INPUT
	Periodic 		: BOOL;
	MasterAbsolute 	: BOOL;
	SlaveAbsolute 	: BOOL;
	CamTable 		: MC_CAM_REF;
END_VAR
END_METHOD

END_INTERFACE

// Examples/CamGearExample
PROGRAM CamGearExample
VAR
	// Hardware definitions
	TcMasterDrive 	: TcAxis_Tc2_MC2;
	TcCamDrive 		: TcAxis_Tc2_MC2;
	TcGearDrive 	: TcAxis_Tc2_MC2;
	
	
	MasterDrive 	: itfAxis;
	CamDrive 		: itfAxis;
	GearDrive 		: itfAxis;
	Table 			: TcCamTable;
	TableData 		: MC_CAM_REF;
	Velocity 		: REAL := 5;
	
	// States
	MasterState 	: INT := 0;
	CamState 		: INT := 0;
	GearState 		: INT := 0;
	
	// Control
	Start 			: BOOL := FALSE;
	
	// Commands
	MasterMove 		: itfCommand;
	TableSet 		: itfCommand;
	CamMove 		: itfSynchronizedAxisCommand;
	GearMove 		: itfSynchronizedAxisCommand;
END_VAR


MasterDrive:= TcMasterDrive;
CamDrive := TcCamDrive;
GearDrive := TcGearDrive;

CASE MasterState OF
	0: // Disabled
		IF Start THEN
			MasterState := MasterState + 1;
		END_IF
		
	1: // Power On
		MasterDrive.Power(Enable:=TRUE, EnablePositive:=TRUE, EnableNegative:=TRUE);
		IF MasterDrive.Status = AXIS_STATUS.Standstill THEN
			MasterState := MasterState + 1;
		END_IF
		
	2: // Wait for other drives 
		IF CamMove.InSync AND GearMove.InSync THEN
			MasterMove := MasterDrive.MoveVelocity(Velocity:=Velocity, Acceleration:=0, Deceleration:=0, Jerk:=0, Direction:=MC_Direction.mcPositiveDirection, BufferMode:=MC_BUFFER_MODE.mcAborting);
			MasterState := MasterState + 1;
		END_IF
		
	3: // Moving
		IF NOT Start THEN
			MasterMove:= MasterDrive.Halt(Deceleration:=0, Jerk:=0, BufferMode:=MC_BUFFER_MODE.mcAborting);
			MasterState := MasterState + 1;
		END_IF
		
	4: // Stopping
		IF NOT MasterMove.Done THEN
			MasterState := MasterState + 1;
		END_IF
		
	5: // Power off
		MasterDrive.Power(Enable:=FALSE, EnablePositive:=FALSE, EnableNegative:=FALSE);
		IF MasterDrive.Status = AXIS_STATUS.Disabled THEN
			MasterState := 0;
		END_IF
END_CASE

CASE CamState OF
	0: // Disabled
		IF Start THEN
			CamState := CamState + 1;
		END_IF
		
	1: // Power On
		CamDrive.Power(Enable:=TRUE, EnablePositive:=TRUE, EnableNegative:=TRUE);
		IF CamDrive.Status = AXIS_STATUS.Standstill AND MasterDrive.Status = AXIS_STATUS.Standstill THEN
			TableSet := Table.Select(CamTable:=TableData, Periodic:=TRUE, MasterAbsolute:=TRUE, SlaveAbsolute:=TRUE);
			CamState := CamState + 1;
		END_IF
		
	2: // Set CAM Table
		IF TableSet.Done THEN
			CamMove := CamDrive.CamIn(Master:=MasterDrive, MasterOffset:=0, SlaveOffset:=0, MasterScaling:=1, SlaveScaling:=1, MasterStartDistance:=0, MasterSyncPosition:=0, 
				StartMode:=MC_StartMode.mcRelative, MasterValueSource:=MC_Source.mcSetValue,CamTable:=Table, BufferMode:=MC_BUFFER_MODE.mcAborting);
			CamState := CamState + 1;
		END_IF
		
	3: // Synchronized
		IF NOT Start THEN
			CamDrive.Release();
			CamState := CamState + 1;
		END_IF
		
	4: // Power off
		CamDrive.Power(Enable:=FALSE, EnablePositive:=FALSE, EnableNegative:=FALSE);
		IF CamDrive.Status = AXIS_STATUS.Disabled THEN
			CamState := 0;
		END_IF
END_CASE

CASE GearState OF
	0: // Disabled
		IF Start THEN
			GearState := GearState + 1;
		END_IF
		
	1: // Power On
		GearDrive.Power(Enable:=TRUE, EnablePositive:=TRUE, EnableNegative:=TRUE);
		IF GearDrive.Status = AXIS_STATUS.Standstill AND MasterDrive.Status = AXIS_STATUS.Standstill THEN
			GearMove := GearDrive.GearIn(Master:=MasterDrive, Ratio:=2, MasterValueSource:=MC_Source.mcSetValue,Acceleration:=0, Deceleration:=0, Jerk:=0, BufferMode:=MC_BUFFER_MODE.mcAborting);
			GearState := GearState + 1;
		END_IF
		
	2: // Synchronized
		IF NOT Start THEN
			GearDrive.Release();
			GearState := GearState + 1;
		END_IF
		
	3: // Power off
		GearDrive.Power(Enable:=FALSE, EnablePositive:=FALSE, EnableNegative:=FALSE);
		IF GearDrive.Status = AXIS_STATUS.Disabled THEN
			GearState := 0;
		END_IF
END_CASE

END_PROGRAM

// TwinCAT Library Template/VendorImplementation/TcAxis_Tc2_MC2
FUNCTION_BLOCK TcAxis_Tc2_MC2 IMPLEMENTS itfAxis
//VAR_INPUT
//	Axis 				: Tc2_MC2.AXIS_REF;
//END_VAR
//VAR_OUTPUT
//END_VAR
VAR_IN_OUT 
	Axis 				: Tc2_MC2.AXIS_REF;
END_VAR
VAR	
	_PowerOn : BOOL;
//	itfCommand      : itfCommand;

//	_fbCommand       	: TcCommand;
	
	_fbAxisCommand   	: TcAxisCommand;

//itfAxisCommand  : itfAxisCommand;
//_Command         : ST_Command;
	

MC : ST_MC;	

count_delete : INT;	
END_VAR

 ACT_Cyclic_Update();

{warning 'add property implementation'}
PROPERTY ActualPosition : REAL
GET
//Actual Position
IF Axis.Status.OpMode.Modulo THEN
    ActualPosition := Axis.NcToPlc.ModuloActPos;
ELSE
    ActualPosition := Axis.NcToPlc.ActPos;
END_IF

count_delete  := count_delete + 1;
END_GET
END_PROPERTY

{warning 'add property implementation'}
PROPERTY ActualTorque : REAL
GET
ActualTorque := Axis.NcToPlc.ActTorque;

count_delete  := count_delete + 1;
END_GET
END_PROPERTY

{warning 'add property implementation'}
PROPERTY ActualVelocity : REAL
GET
//Actual Velocity
ActualVelocity := Axis.NcToPlc.ActVelo;
END_GET
END_PROPERTY

{attribute 'TcRpcEnable'}
METHOD Power 		: itfCommand
VAR_INPUT
	Enable			: BOOL;
	EnablePositive	: BOOL;
	EnableNegative	: BOOL;
END_VAR
VAR
	_fbCommand       	: TcCommand;
	itfCommand      : itfCommand;
	Command         : ST_Command;
END_VAR

itfCommand := _fbCommand;

MC.Power(
	Axis:= Axis, 
	Enable:= Enable, 
	Enable_Positive:= EnablePositive, 
	Enable_Negative:= EnableNegative, 
	Override:= 100, 
	BufferMode:= , 
	Options:= , 
	Status=> , 
	Busy=> Command.Busy,
	Active=> Command.Active,
	Error=> Command.Error,
	ErrorID=> Command.ErrorID_Udint);
		
itfCommand.Busy   		:=	Command.Busy;
itfCommand.Active 		:=	Command.Active;
itfCommand.Error 		:=	Command.Error;
itfCommand.ErrorID_Udint :=	Command.ErrorID_Udint;
	
Power := itfCommand;

_PowerOn := MC.Power.Enable;
END_METHOD

{warning 'add method implementation '}
METHOD ReadBoolParameter 	: MC_Error
VAR_INPUT
	ParameterNumber			: INT;
END_VAR
VAR_OUTPUT
	Value					: BOOL;
END_VAR
VAR
	fbReadBoolParameter 	: Tc2_MC2.MC_ReadBoolParameter;
END_VAR

fbReadBoolParameter(
	Axis:= Axis, 
	Enable:= TRUE, 
	ParameterNumber:= ParameterNumber, 
	ReadMode:= , 
	Valid=> , 
	Busy=> , 
	Error=> , 
	ErrorID=> , 
	Value=> Value);


count_delete  := count_delete + 1;
END_METHOD

{warning 'add method implementation '}
METHOD ReadParameter 	: MC_Error
VAR_INPUT
	ParameterNumber		: INT;
END_VAR
VAR_OUTPUT
	Value				: REAL;
END_VAR
VAR
	fbReadParameter		: Tc2_MC2.MC_ReadParameter;
END_VAR

fbReadParameter(
	Axis:= Axis, 
	Enable:= TRUE, 
	ParameterNumber:= ParameterNumber, 
	ReadMode:= , 
	Valid=> , 
	Busy=> , 
	Error=> , 
	ErrorID=> , 
	Value=> Value);


count_delete  := count_delete + 1;
END_METHOD

{warning 'add method implementation '}
METHOD Release : MC_Error

VAR
	
END_VAR
count_delete  := count_delete + 1;
END_METHOD

{attribute 'TcRpcEnable'}
METHOD Reset 		: itfCommand

VAR
	fbReset 		: Tc2_MC2.MC_RESET;
END_VAR

fbReset(
	Axis:= Axis, 
	Execute:= TRUE, 
	Done=> , 
	Busy=> , 
	Error=> , 
	ErrorID=> );


count_delete  := count_delete + 1;
END_METHOD

{warning 'add method implementation '}
METHOD SetOverride 	: MC_Error
VAR_INPUT
	VelFactor		: REAL;
	AccFactor		: REAL;
	JerkFactor		: REAL;
END_VAR

VAR
	fbSetOverride 	: Tc2_MC2.MC_SetOverride;
END_VAR

fbSetOverride(
	Axis:= Axis, 
	Enable:= TRUE, 
	VelFactor:= VelFactor, 
	AccFactor:= AccFactor, 
	JerkFactor:= JerkFactor, 
	Enabled=> , 
	Busy=> , 
	Error=> , 
	ErrorID=> );

count_delete  := count_delete + 1;
END_METHOD

{warning 'add method implementation '}
METHOD SetPosition 	: itfCommand
VAR_INPUT
	Position		: REAL;
	Relative		: BOOL; (* RELATIVE=True, ABSOLUTE=False (Default)*)
//	ExecutionMode	: MC_ExecutionMode;
    ExecutionMode	: Tc2_MC2.ST_SetPositionOptions;
END_VAR

VAR
	fbSetPosition 	: Tc2_MC2.MC_SetPosition;
END_VAR

fbSetPosition(
	Axis:= Axis, 
	Execute:= TRUE, 
	Position:= Position, 
	Mode:= Relative, 
	Options:= ExecutionMode, 
	Done=> , 
	Busy=> , 
	Error=> , 
	ErrorID=> );

count_delete  := count_delete + 1;
END_METHOD

{warning 'add method implementation '}
METHOD WriteBoolParameter 	: MC_Error
VAR_INPUT
	ParameterNumber			: INT;
	Value					: BOOL;
END_VAR

VAR
	fbWriteBoolParameter 	: Tc2_MC2.MC_WriteBoolParameter;	
END_VAR

fbWriteBoolParameter(
	Axis:= Axis, 
	Execute:= TRUE, 
	ParameterNumber:= ParameterNumber, 
	Value:= Value, 
	Done=> , 
	Busy=> , 
	Error=> , 
	ErrorID=> );

count_delete  := count_delete + 1;
END_METHOD

{warning 'add method implementation '}
METHOD WriteParameter 	: MC_Error
VAR_INPUT
	ParameterNumber		: INT;
	Value				: REAL;
END_VAR

VAR
	fbWriteParameter 	: Tc2_MC2.MC_WriteParameter;	
END_VAR

fbWriteParameter(
	Axis:= Axis, 
	Execute:= TRUE, 
	ParameterNumber:= ParameterNumber, 
	Value:= Value, 
	Done=> , 
	Busy=> , 
	Error=> , 
	ErrorID=> );

count_delete  := count_delete + 1;
END_METHOD

{warning 'add method implementation '}
METHOD CombineAxes 			: itfSynchronizedAxisCommand
VAR_INPUT
	Master1					: itfAxis;
	Master2					: itfAxis;
	CombineMode				: MC_COMBINE_MODE;
	GearRatioNumeratorM1	: INT;
	GearRatioDenominatorM1	: INT;
	GearRatioNumeratorM2	: INT;
	GearRatioDenominatorM2	: INT;
	MasterValueSourceM1		: MC_SOURCE;
	MasterValueSourceM2		: MC_SOURCE;
	BufferMode				: MC_BUFFER_MODE;
END_VAR
VAR
	
END_VAR

//fbGearIn(
//	Master:= , 
//	Slave:= , 
//	Execute:= , 
//	RatioNumerator:= , 
//	RatioDenominator:= , 
//	Acceleration:= , 
//	Deceleration:= , 
//	Jerk:= , 
//	BufferMode:= , 
//	Options:= , 
//	InGear=> , 
//	Busy=> , 
//	Active=> , 
//	CommandAborted=> , 
//	Error=> , 
//	ErrorID=> );


count_delete  := count_delete + 1;
END_METHOD

{attribute 'TcRpcEnable'}
METHOD GearIn 			: itfSynchronizedAxisCommand
VAR_INPUT
//	Master				: itfAxis;
//	Master				: Tc2_MC2.AXIS_REF;
//	Slave				: Tc2_MC2.AXIS_REF;		
//	Ratio				: REAL;
//	MasterValueSource	: INT;
	RatioNumerator		: LREAL;
	RatioDenominator	: UINT;
	Acceleration		: REAL;
	Deceleration		: REAL;
	Jerk				: REAL;
	BufferMode			: MC_BUFFER_MODE;
//	BufferMode			: Tc2_MC2.MC_BufferMode;
//	Options             : Tc2_MC2.ST_GearInOptions;
END_VAR
VAR_IN_OUT 
	Slave				: Tc2_MC2.AXIS_REF;	
END_VAR
VAR
	fbGearIn			: Tc2_MC2.MC_GearIn;	
END_VAR
	
fbGearIn(
	Master:= Axis, 
	Slave:= Slave, 
	Execute:= TRUE, 
	RatioNumerator:= RatioNumerator, 
	RatioDenominator:= RatioDenominator, 
	Acceleration:= ,//Acceleration, 
	Deceleration:= ,//Deceleration, 
	Jerk:= ,//Jerk, 
	BufferMode:= ,//BufferMode,//BufferMode, 
	Options:= ,//Options, 
	InGear=> ,//Geared , 
	Busy=> , 
	Active=> , 
	CommandAborted=> , 
	Error=> , 
	ErrorID=> );

count_delete  := count_delete + 1;
END_METHOD

{warning 'add method implementation '}
METHOD PhasingAbsolute 	: itfSynchronizedAxisCommand
VAR_INPUT
//	Master				: itfAxis;
	Master				: Tc2_MC2.AXIS_REF;
	Slave				: Tc2_MC2.AXIS_REF;		
	PhaseShift			: REAL;
	Velocity			: REAL;
	Acceleration		: REAL;
	Deceleration		: REAL;
	Jerk				: REAL;
	BufferMode			: MC_BUFFER_MODE;
END_VAR
VAR
	fbPhasingAbsolute	: Tc2_MC2.MC_PhasingAbsolute;
END_VAR

fbPhasingAbsolute(
	Master:= Master, 
	Slave:= Slave, 
	Execute:= TRUE, 
	ContinuousUpdate:= , 
	PhaseShift:= , 
	Velocity:= , 
	Acceleration:= , 
	Deceleration:= , 
	Jerk:= , 
	BufferMode:= , 
	Options:= , 
	Done=> , 
	Busy=> , 
	Active=> , 
	CommandAborted=> , 
	Error=> , 
	ErrorID=> , 
	AbsolutePhaseShift=> );

count_delete  := count_delete + 1;
END_METHOD

{warning 'add method implementation '}
METHOD PhasingRelative 	: itfSynchronizedAxisCommand
VAR_INPUT
//	Master				: itfAxis;
	Master				: Tc2_MC2.AXIS_REF;
	Slave				: Tc2_MC2.AXIS_REF;		
	PhaseShift			: REAL;
	Velocity			: REAL;
	Acceleration		: REAL;
	Deceleration		: REAL;
	Jerk				: REAL;
	BufferMode			: MC_BUFFER_MODE;
END_VAR
VAR
	fbPhasingRelative	: Tc2_MC2.MC_PhasingRelative;
END_VAR


fbPhasingRelative(
	Master:= Master, 
	Slave:= Slave, 
	Execute:= , 
	ContinuousUpdate:= , 
	PhaseShift:= , 
	Velocity:= , 
	Acceleration:= , 
	Deceleration:= , 
	Jerk:= , 
	BufferMode:= , 
	Options:= , 
	Done=> , 
	Busy=> , 
	Active=> , 
	CommandAborted=> , 
	Error=> , 
	ErrorID=> , 
	CoveredPhaseShift=> );

count_delete  := count_delete + 1;
END_METHOD

{warning 'add method implementation '}
METHOD AccelerationProfile 	: itfCommand
VAR_INPUT
	TimeScale				: REAL;
	AccelerationScale		: REAL;
	Offset					: REAL;
	BufferMode				: MC_BUFFER_MODE;
END_VAR
VAR
	
END_VAR
count_delete  := count_delete + 1;
END_METHOD

{warning 'add method implementation '}
METHOD Halt 		: itfAxisCommand
VAR_INPUT
	Deceleration	: REAL;
	Jerk			: REAL;
	BufferMode		: MC_BUFFER_MODE;
END_VAR
VAR
	fbHalt			: Tc2_MC2.MC_HALT;
END_VAR

fbHalt(
	Axis:= Axis, 
	Execute:= , 
	Deceleration:= Deceleration, 
	Jerk:= Jerk, 
	BufferMode:= , //BufferMode, 
	Options:= , 
	Done=> , 
	Busy=> , 
	Active=> , 
	CommandAborted=> , 
	Error=> , 
	ErrorID=> );

count_delete  := count_delete + 1;
END_METHOD

{warning 'add method implementation '}
METHOD HaltSuperimposed : itfAxisCommand
VAR_INPUT
	Deceleration		: REAL;
	Jerk				: REAL;
END_VAR
VAR
	
END_VAR
count_delete  := count_delete + 1;
END_METHOD

{warning 'add method implementation '}
METHOD Home 		: itfAxisCommand
VAR_INPUT
	Position		: REAL;
	Velocity		: REAL;
	EndVelocity		: REAL;
	Acceleration	: REAL;
	Deceleration	: REAL;
	Jerk			: REAL;
	Direction		: MC_Direction;
	HomingMode		: INT;
	BufferMode		: MC_BUFFER_MODE;
END_VAR
VAR
	fbHome			: Tc2_MC2.MC_HOME;
END_VAR

fbHome(
	Axis:= Axis, 
	Execute:= TRUE, 
	Position:= Position, 
	HomingMode:= HomingMode, 
	BufferMode:= ,//BufferMode , 
	Options:= , 
	bCalibrationCam:= , 
	Done=> , 
	Busy=> , 
	Active=> , 
	CommandAborted=> , 
	Error=> , 
	ErrorID=> );

count_delete  := count_delete + 1;
END_METHOD

{warning 'add method implementation '}
METHOD Jog 			: itfAxisCommand
VAR_INPUT
    JogForward 		: BOOL;
    JogBackwards 	: BOOL;
    Mode     		: Tc2_MC2.E_JogMode;
    Position        : LREAL;
    Velocity        : LREAL;
    Acceleration 	: LREAL;
    Deceleration 	: LREAL;
    Jerk     		: LREAL;
END_VAR
VAR
	fbJog			: Tc2_MC2.MC_JOG;
END_VAR

count_delete  := count_delete + 1;
END_METHOD

{attribute 'TcRpcEnable'}
METHOD MoveAbsolute : itfAxisCommand
VAR_INPUT
	Position		: REAL;
	Velocity		: REAL;
	Acceleration	: REAL;
	Deceleration	: REAL;
	Jerk			: REAL;
	Direction		: MC_Direction;
	BufferMode		: MC_BUFFER_MODE;
END_VAR

VAR
	itfAxisCommand   : itfAxisCommand;
    _Command         : ST_Command;
END_VAR
itfAxisCommand := _fbAxisCommand;
	
MC.MoveAbsolute(
	Axis:= Axis, 
	Execute:= TRUE ,
	Position:= Position, 
	Velocity:= Velocity, 
	Acceleration:= Acceleration, 
	Deceleration:= Deceleration, 
	Jerk:= Jerk, 
	BufferMode:= BufferMode,//BufferMode, 
	Options:= , 
	Done=> _Command.Done, 
	Busy=> _Command.Busy, 
	Active=>_Command.Active, 
	CommandAborted=> _Command.CommandAborted, 
	Error=> _Command.Error, 
	ErrorID=> _Command.ErrorID_Udint);
	
MC.MoveAbsolute(
	Axis:= Axis, 
	Execute:= FALSE);	

itfAxisCommand.Done 				:=  _Command.Done AND ActualPosition = Position;             
itfAxisCommand.Busy   				:=	_Command.Busy;
itfAxisCommand.Active 				:=	_Command.Active;
itfAxisCommand.CommandAborted		:=	_Command.CommandAborted;
itfAxisCommand.Error 				:=	_Command.Error;
itfAxisCommand.ErrorID_Udint 		:=	_Command.ErrorID_Udint;

MoveAbsolute := itfAxisCommand;
END_METHOD

{warning 'add method implementation '}
METHOD MoveAdditive : itfAxisCommand
VAR_INPUT
	Distance		: REAL;
	Velocity		: REAL;
	Acceleration	: REAL;
	Deceleration	: REAL;
	Jerk			: REAL;
	BufferMode		: MC_BUFFER_MODE;
END_VAR
VAR
	fbMoveAdditive 	: Tc2_MC2.MC_MoveAdditive;	
END_VAR

fbMoveAdditive(
	Axis:= Axis, 
	Execute:= TRUE, 
	Distance:= Distance, 
	Velocity:= Velocity, 
	Acceleration:= Acceleration, 
	Deceleration:= Deceleration, 
	Jerk:= Jerk, 
	BufferMode:= , //BufferMode, 
	Options:= , 
	Done=> , 
	Busy=> , 
	Active=> , 
	CommandAborted=> , 
	Error=> , 
	ErrorID=> );


count_delete  := count_delete + 1;
END_METHOD

{warning 'add method implementation '}
METHOD MoveContinuousAbsolute 	: itfContinuousAxisCommand
VAR_INPUT
	Position					: REAL;
	EndVelocity					: REAL;
	Velocity					: REAL;
	Acceleration				: REAL;
	Deceleration				: REAL;
	Jerk						: REAL;
	Direction					: MC_DIRECTION;
	BufferMode					: MC_BUFFER_MODE;
END_VAR
VAR
	fbMoveContinuousAbsolute 	: Tc2_MC2.MC_MoveContinuousAbsolute;		
END_VAR

fbMoveContinuousAbsolute(
	Axis:= Axis, 
	Execute:= TRUE, 
	Position:= Position, 
	Velocity:= Velocity, 
	EndVelocity:= EndVelocity, 
	Acceleration:= Acceleration, 
	Deceleration:= Deceleration, 
	Jerk:= Jerk, 
	BufferMode:= ,//BufferMode, 
	Options:= , 
	InEndVelocity=> , 
	Busy=> , 
	Active=> , 
	CommandAborted=> , 
	Error=> , 
	ErrorID=> );


count_delete  := count_delete + 1;
END_METHOD

{warning 'add method implementation '}
METHOD MoveContinuousRelative 	: itfContinuousAxisCommand
VAR_INPUT
	Distance					: REAL;
	EndVelocity					: REAL;
	Velocity					: REAL;
	Acceleration				: REAL;
	Deceleration				: REAL;
	Jerk						: REAL;
	Direction					: MC_DIRECTION;
	BufferMode					: MC_BUFFER_MODE;
END_VAR
VAR
	fbMoveContinuousRelative 	: Tc2_MC2.MC_MoveContinuousRelative;
END_VAR

fbMoveContinuousRelative(
	Axis:= Axis, 
	Execute:= TRUE, 
	Distance:= Distance, 
	Velocity:= Velocity, 
	EndVelocity:= EndVelocity, 
	Acceleration:= Acceleration, 
	Deceleration:= Deceleration, 
	Jerk:= Jerk, 
	BufferMode:= ,//BufferMode, 
	Options:= , 
	InEndVelocity=> , 
	Busy=> , 
	Active=> , 
	CommandAborted=> , 
	Error=> , 
	ErrorID=> );



count_delete  := count_delete + 1;
END_METHOD

{attribute 'TcRpcEnable'}
METHOD MoveRelative 	: itfAxisCommand
VAR_INPUT
	Distance			: REAL;
	Velocity			: REAL;
	Acceleration		: REAL;
	Deceleration		: REAL;
	Jerk				: REAL;
	BufferMode			: MC_BUFFER_MODE;
END_VAR
VAR
	itfAxisCommand   : itfAxisCommand;
	_Command         : ST_Command;
END_VAR
itfAxisCommand := _fbAxisCommand;

MC.MoveRelative(
	Axis:= Axis, 
	Execute:= TRUE, 
	Distance:= Distance, 
	Velocity:= Velocity, 
	Acceleration:= Acceleration, 
	Deceleration:= Deceleration, 
	Jerk:= Jerk, 
	BufferMode:= ,//BufferMode, 
	Options:= , 
	Done=> _Command.Done, 
	Busy=> _Command.Busy, 
	Active=> _Command.Active, 
	CommandAborted=> _Command.CommandAborted, 
	Error=> _Command.Error, 
	ErrorID=> _Command.ErrorID_Udint);
	
MC.MoveRelative(
	Axis:= Axis, 
	Execute:= FALSE);		
	
itfAxisCommand.Done 				:=  _Command.Done; //AND ActualPosition = ActualPosition + Distance;             
itfAxisCommand.Busy   				:=	_Command.Busy;
itfAxisCommand.Active 				:=	_Command.Active;
itfAxisCommand.CommandAborted		:=	_Command.CommandAborted;
itfAxisCommand.Error 				:=	_Command.Error;
itfAxisCommand.ErrorID_Udint 		:=	_Command.ErrorID_Udint;

MoveRelative := itfAxisCommand;
END_METHOD

{warning 'add method implementation '}
METHOD MoveSuperimposed 	: itfAxisCommand
VAR_INPUT
	Distance				: REAL;
	VelocityDiff			: REAL;
	Acceleration			: REAL;
	Deceleration			: REAL;
	Jerk					: REAL;
END_VAR
VAR
	fbMoveSuperimposed	 	: Tc2_MC2.MC_MoveSuperimposed;	
END_VAR

fbMoveSuperimposed(
	Axis:= Axis, 
	Execute:= TRUE, 
	Mode:= , 
	Distance:= , 
	VelocityDiff:= VelocityDiff, 
	Acceleration:= Acceleration, 
	Deceleration:= Deceleration, 
	Jerk:= Jerk, 
	VelocityProcess:= , 
	Length:= , 
	Options:= , 
	Done=> , 
	Busy=> , 
	Active=> , 
	CommandAborted=> , 
	Error=> , 
	ErrorID=> , 
	Warning=> , 
	WarningId=> , 
	ActualVelocityDiff=> , 
	ActualDistance=> , 
	ActualLength=> , 
	ActualAcceleration=> , 
	ActualDeceleration=> );

count_delete  := count_delete + 1;
END_METHOD

{warning 'add method implementation '}
METHOD MoveVelocity 	: itfContinuousAxisCommand
VAR_INPUT
	Velocity			: REAL;
	Acceleration		: REAL;
	Deceleration		: REAL;
	Jerk				: REAL;
	Direction			: MC_Direction;
	BufferMode			: MC_BUFFER_MODE;
END_VAR
VAR
	fbMoveVelocity	 	: Tc2_MC2.MC_MoveVelocity;	
END_VAR

fbMoveVelocity(
	Axis:= Axis, 
	Execute:= TRUE, 
	Velocity:= Velocity, 
	Acceleration:= Acceleration, 
	Deceleration:= Deceleration, 
	Jerk:= Jerk, 
	Direction:= Direction, 
	BufferMode:= , //BufferMode
	Options:= , 
	InVelocity=> , 
	Busy=> , 
	Active=> , 
	CommandAborted=> , 
	Error=> , 
	ErrorID=> );	

count_delete  := count_delete + 1;
END_METHOD

{warning 'add method implementation '}
METHOD PositionProfile 	: itfCommand
VAR_INPUT
	TimeScale			: REAL;
	PositionScale		: REAL;
	Offset				: REAL;
	BufferMode			: MC_BUFFER_MODE;
END_VAR
VAR
//	fbPositionProfile	 	: Tc2_MC2.;	
END_VAR






count_delete  := count_delete + 1;
END_METHOD

{warning 'add method implementation '}
METHOD Stop 		: itfAxisCommand
VAR_INPUT
	Deceleration	: REAL;
	Jerk			: REAL;
END_VAR
VAR
	fbStop			: Tc2_MC2.MC_STOP;
END_VAR

fbStop(
	Axis:= Axis, 
	Execute:= TRUE, 
	Deceleration:= Deceleration, 
	Jerk:= Jerk, 
	Options:= , 
	Done=> , 
	Busy=> , 
	Active=> , 
	CommandAborted=> , 
	Error=> , 
	ErrorID=> );

count_delete  := count_delete + 1;
END_METHOD

{warning 'add method implementation '}
METHOD TorqueControl 	: itfAxisCommand
VAR_INPUT
	Torque				: REAL;
	TorqueRamp			: REAL;
	Velocity			: REAL;
	Acceleration		: REAL;
	Deceleration		: REAL;
	Jerk				: REAL;
	Direction			: MC_DIRECTION;
	BufferMode			: MC_BUFFER_MODE;
END_VAR
VAR
	fbTorqueControl		: Tc2_MC2.MC_TorqueControl;
END_VAR

fbTorqueControl(
	Axis:= Axis, 
	Execute:= , 
	ContinuousUpdate:= , 
	Relative:= , 
	Torque:= Torque, 
	TorqueRamp:= TorqueRamp, 
	VelocityLimitHigh:= , 
	VelocityLimitLow:= , 
	BufferMode:= , 
	Options:= , 
	InTorque=> , 
	Busy=> , 
	Active=> , 
	CommandAborted=> , 
	Error=> , 
	ErrorId=> );

count_delete  := count_delete + 1;
END_METHOD

{warning 'add method implementation '}
METHOD VelocityProfile 	: itfCommand
VAR_INPUT
	TimeScale			: REAL;
	VelocityScale		: REAL;
	Offset				: REAL;
	BufferMode			: MC_BUFFER_MODE;
END_VAR
VAR
	
END_VAR
count_delete  := count_delete + 1;
END_METHOD

{warning 'add property implementation'}
PROPERTY AxisWarning : BOOL
GET
count_delete  := count_delete + 1;
END_GET
END_PROPERTY

{warning 'add property implementation'}
PROPERTY CommunicationReady : BOOL
GET
count_delete  := count_delete + 1;
END_GET
END_PROPERTY

{warning 'add property implementation'}
PROPERTY Direction : AXIS_DIRECTION
GET
count_delete  := count_delete + 1;
END_GET
END_PROPERTY

PROPERTY Error : BOOL
GET
Error :=  Axis.Status.Error;
END_GET
END_PROPERTY

{warning 'add property implementation'}
PROPERTY ErrorId : WORD
GET

//ErrorId := Axis.Status.ErrorID;

count_delete  := count_delete + 1;
END_GET
END_PROPERTY

PROPERTY ErrorId_Udint_Status : UDINT
GET
ErrorId_Udint_Status := Axis.Status.ErrorID;
END_GET
END_PROPERTY

PROPERTY Geared : BOOL
GET
Geared :=  Axis.Status.Coupled;
//Axis.NcToPlc.CoupleState
END_GET
END_PROPERTY

{warning 'add property implementation'}
PROPERTY HomeAbsSwitch : BOOL
GET
count_delete  := count_delete + 1;
END_GET
END_PROPERTY


PROPERTY IsHomed : BOOL
GET

IsHomed := Axis.Status.Homed;
END_GET
END_PROPERTY

{warning 'add property implementation'}
PROPERTY LimitSwitchNegative : BOOL
GET

LimitSwitchNegative := Axis.Status.SoftLimitMinExceeded;

count_delete  := count_delete + 1;
END_GET
END_PROPERTY

{warning 'add property implementation'}
PROPERTY LimitSwitchPositive : BOOL
GET

LimitSwitchPositive := Axis.Status.SoftLimitMaxExceeded;

count_delete  := count_delete + 1;
END_GET
END_PROPERTY

{warning 'add property implementation'}
PROPERTY MotionStatus : MOTION_STATUS
GET
END_GET
END_PROPERTY

{attribute ‘monitoring’ := ‘call’}
PROPERTY PowerOn : BOOL
GET
PowerOn := _PowerOn;
END_GET
END_PROPERTY

{warning 'add property implementation'}
PROPERTY ReadyForPowerOn : BOOL
GET
count_delete  := count_delete + 1;
END_GET
END_PROPERTY

{warning 'add property implementation'}
PROPERTY Simulation : BOOL
GET
count_delete  := count_delete + 1;
END_GET
END_PROPERTY

{attribute ‘monitoring’ := ‘call’}
PROPERTY Status : Tc2_MC2.MC_AxisStates
GET
VAR
//	ReadStatus : Tc2_MC2.MC_ReadStatus;
END_VAR

//ReadStatus(
//	Axis:= Axis, 
//	Enable:= FALSE);

//ReadStatus(
//	Axis:= Axis, 
//	Enable:= TRUE, 
//	Valid=> , 
//	Busy=> , 
//	Error=> , 
//	ErrorID=> , 
//	ErrorStop=>, 
//	Disabled=> , 
//	StandStill=> , 
//	DiscreteMotion=> , 
//	ContinuousMotion=> , 
//	SynchronizedMotion=> , 
//	Homing=> , 
//	ConstantVelocity=> , 
//	Accelerating=> , 
//	Decelerating=> , 
//	Status=> );

Status := Axis.Status.MotionState;
END_GET
END_PROPERTY

ACTION ACT_Cyclic_Update:
//update local variables from hardware
Axis.ReadStatus();
END_ACTION

END_FUNCTION_BLOCK

// TwinCAT Library Template/VendorImplementation/TcCommand
FUNCTION_BLOCK TcCommand IMPLEMENTS itfCommand
//VAR_INPUT
//END_VAR
//VAR_OUTPUT
//END_VAR
VAR
	_Command        : ST_Command;	
END_VAR

{warning 'add method implementation '}
METHOD Abort : MC_Error
VAR
	
END_VAR
END_METHOD

{warning 'add property implementation'}
PROPERTY Active : BOOL
GET
Active := _Command.Active;
END_GET
SET
_Command.Active := Active;
END_SET
END_PROPERTY

{warning 'add property implementation'}
PROPERTY Busy : BOOL
GET
Busy := _Command.Busy;
END_GET
SET
_Command.Busy := Busy;
END_SET
END_PROPERTY

{warning 'add property implementation'}
PROPERTY Command : MC_COMMAND_REF
GET
Command := _Command.Command;
END_GET
SET
 _Command.Command :=  Command;
END_SET
END_PROPERTY

{warning 'add property implementation'}
PROPERTY CommandAborted : BOOL
GET
CommandAborted := _Command.CommandAborted;
END_GET
SET
 _Command.CommandAborted := CommandAborted;
END_SET
END_PROPERTY

{warning 'add property implementation'}
PROPERTY Done : BOOL
GET
Done := _Command.Done;
END_GET
SET
_Command.Done := Done;
END_SET
END_PROPERTY

{warning 'add property implementation'}
PROPERTY Error : BOOL
GET
Error := _Command.Error;
END_GET
SET
_Command.Error := Error;
END_SET
END_PROPERTY

{warning 'add property implementation'}
PROPERTY ErrorId : MC_Error
GET
ErrorId := _Command.ErrorId;
END_GET
SET
_Command.ErrorId := ErrorId;
END_SET
END_PROPERTY

PROPERTY ErrorID_Udint : UDINT
GET
ErrorID_Udint := _Command.ErrorID_Udint;
END_GET
SET
_Command.ErrorID_Udint := ErrorID_Udint;
END_SET
END_PROPERTY

{warning 'add method implementation '}
METHOD Wait : MC_Error (* This method only makes sense in the IEC 61499 environment*)
VAR_INPUT
	Timeout	: TIME;
	AbortOnTimeout	: BOOL;
END_VAR
VAR
	
END_VAR
END_METHOD

END_FUNCTION_BLOCK

// TwinCAT Library Template/VendorImplementation/TcAxisCommand
FUNCTION_BLOCK TcAxisCommand IMPLEMENTS itfAxisCommand
//VAR_INPUT
//END_VAR
//VAR_OUTPUT
//END_VAR
VAR
	_Command        : ST_Command;	
END_VAR

{warning 'Agregar implementación de método'}
METHOD Abort : MC_Error
END_METHOD

{warning 'Agregar implementación de propiedad'}
PROPERTY Active : BOOL
GET
END_GET
SET
END_SET
END_PROPERTY

{warning 'Agregar implementación de propiedad'}
PROPERTY Busy : BOOL
GET
END_GET
SET
END_SET
END_PROPERTY

{warning 'Agregar implementación de propiedad'}
PROPERTY Command : MC_COMMAND_REF
GET
END_GET
SET
END_SET
END_PROPERTY

{warning 'Agregar implementación de propiedad'}
PROPERTY CommandAborted : BOOL
GET
END_GET
SET
END_SET
END_PROPERTY

{warning 'Agregar implementación de propiedad'}
PROPERTY Done : BOOL
GET
Done := _Command.Done;
END_GET
SET
_Command.Done := Done;
END_SET
END_PROPERTY

{warning 'Agregar implementación de propiedad'}
PROPERTY Error : BOOL
GET
END_GET
SET
END_SET
END_PROPERTY

{warning 'Agregar implementación de propiedad'}
PROPERTY ErrorId : MC_Error
GET
END_GET
SET
END_SET
END_PROPERTY

{warning 'Agregar implementación de propiedad'}
PROPERTY ErrorID_Udint : MC_ErrorID_Udint
GET
END_GET
SET
END_SET
END_PROPERTY

{warning 'add method implementation '}
METHOD Update 		: MC_Error
VAR_INPUT
	Position		: REAL;
	Velocity		: REAL;
	EndVelocity		: REAL;
	Acceleration	: REAL;
	Deceleration	: REAL;
	Jerk			: REAL;
END_VAR
END_METHOD

{warning 'Agregar implementación de método'}
METHOD Wait : MC_Error (* This method only makes sense in the IEC 61499 environment*)
VAR_INPUT
	Timeout	: TIME;
	AbortOnTimeout	: BOOL;
END_VAR
END_METHOD

END_FUNCTION_BLOCK

// TwinCAT Library Template/VendorImplementation/TcCamTable
FUNCTION_BLOCK TcCamTable IMPLEMENTS itfCamTable
VAR_INPUT
END_VAR
VAR_OUTPUT
END_VAR
VAR
END_VAR

{warning 'add method implementation '}
METHOD Select 		: itfCommand
VAR_INPUT	
	Periodic		: BOOL;
	MasterAbsolute	: BOOL;
	SlaveAbsolute	: BOOL;
	CamTable		: MC_CAM_REF;
END_VAR
VAR
	
END_VAR
END_METHOD

END_FUNCTION_BLOCK

// Examples/LabelingExample
PROGRAM LabelingExample
VAR
	AXIS_REF_LabelDrive			: TC2_MC2.AXIS_REF;
	AXIS_REF_Conveyor 			: TC2_MC2.AXIS_REF;

	// Hardware definitions
	LabelDrive 			: TcAxis_Tc2_MC2;
	Conveyor 			: TcAxis_Tc2_MC2;
	LabelLength 		: REAL := 100;
	SensorDistance 		: REAL := 10;
	Velocity 			: REAL := 5;
	ProductDetection 	: BOOL := FALSE;
	DelayTimer 			: TON;
	
	// States
	ConveyorState 		: INT := 0;
	LabelDriveState 	: INT := 0;
	
	// Control
	Start 				: BOOL := FALSE;
	
	// Commands
	ConveyorMove 		: itfCommand;
	LabelDriveMove 		: itfCommand;
END_VAR


LabelDrive(Axis:= AXIS_REF_LabelDrive);
Conveyor(Axis:= AXIS_REF_Conveyor);

// Run the timer. As it is a classic FB it should be called every cycle
DelayTimer(IN:=ProductDetection, PT:= INT_TO_TIME(REAL_TO_INT(SensorDistance * 1000 / Velocity)));

CASE ConveyorState OF
	0: // Disabled
		IF Start THEN
			ConveyorState := ConveyorState + 1;
		END_IF
		
	1: // Power On
		Conveyor.Power(Enable:=TRUE, EnablePositive:=TRUE, EnableNegative:=TRUE);
		//IF Conveyor.Status = AXIS_STATUS.Standstill THEN
	  IF Conveyor.Status = Tc2_MC2.MC_AXISSTATE_STANDSTILL THEN
			ConveyorState := ConveyorState + 1;
		END_IF
		
	2: // Wait for LabelDrive 
		//IF LabelDrive.Status = AXIS_STATUS.Standstill THEN
		IF LabelDrive.Status =  Tc2_MC2.MC_AXISSTATE_STANDSTILL THEN
			ConveyorMove := Conveyor.MoveVelocity(Velocity:=Velocity, Acceleration:=0, Deceleration:=0, Jerk:=0, Direction:=MC_Direction.mcPositiveDirection, BufferMode:=MC_BUFFER_MODE.mcAborting);
			ConveyorState := ConveyorState + 1;
		END_IF
		
	3: // Moving
		IF NOT Start THEN
			ConveyorMove := Conveyor.Halt(Deceleration:=0, Jerk:=0, BufferMode:=MC_BUFFER_MODE.mcAborting);
			ConveyorState := ConveyorState + 1;
		END_IF
		
	4: // Stopping
		IF ConveyorMove.Done THEN
			ConveyorState := ConveyorState + 1;
		END_IF
		
	5: // Power off
		Conveyor.Power(Enable:=FALSE, EnablePositive:=FALSE, EnableNegative:=FALSE);
		IF Conveyor.Status = AXIS_STATUS.Disabled THEN
			ConveyorState := 0;
		END_IF
END_CASE

CASE LabelDriveState OF
	0: // Disabled
		IF Start THEN
			LabelDriveState := LabelDriveState + 1;
		END_IF
		
	1: // Power On
		LabelDrive.Power(Enable:=TRUE, EnablePositive:=TRUE, EnableNegative:=TRUE);
		//IF LabelDrive.Status = AXIS_STATUS.Standstill THEN
		IF LabelDrive.Status = Tc2_MC2.MC_AXISSTATE_STANDSTILL THEN
			LabelDriveState := LabelDriveState + 1;
		END_IF
		
	2: // Wait for Conveyor 
		//IF Conveyor.Status = AXIS_STATUS.Standstill THEN
		IF Conveyor.Status = Tc2_MC2.MC_AXISSTATE_STANDSTILL THEN
			LabelDriveState := LabelDriveState + 1;
		END_IF
						
	3: // Wait for product
		IF NOT Start THEN
			LabelDriveState := 5;
		END_IF
		IF DelayTimer.Q THEN
			LabelDriveMove := LabelDrive.MoveRelative(Distance:=LabelLength, Velocity:=Velocity, Acceleration:=0, Deceleration:=0, Jerk:=0, BufferMode:=MC_BUFFER_MODE.mcAborting);
			LabelDriveState := LabelDriveState + 1;
		END_IF
		
	4: // Wait for label to be transfered
		IF LabelDriveMove.Done AND NOT DelayTimer.Q THEN
			LabelDriveState := 3;
		END_IF
		
	5: // Power off
		Conveyor.Power(Enable:=FALSE, EnablePositive:=FALSE, EnableNegative:=FALSE);
		IF Conveyor.Status = AXIS_STATUS.Disabled THEN
			LabelDriveState := 0;
		END_IF
	
END_CASE

END_PROGRAM

// Examples/MAIN_Examples
PROGRAM MAIN_Examples
VAR
//	fbAxis_X1 				: TcAxis_Tc2_MC2;
			
	fbSum : FB_Sum;
END_VAR


WareHousingExample();

LabelingExample();

//CamGearExample();

END_PROGRAM

// Examples/WareHousingExample
PROGRAM WareHousingExample
VAR
		stateOOP 				: INT;
		stepOn 					: BOOL := FALSE;
                            	
		AXIS_REF_X1 			: Tc2_MC2.AXIS_REF;
		AXIS_REF_Y 				: Tc2_MC2.AXIS_REF;
		AXIS_REF_Z 				: Tc2_MC2.AXIS_REF;
		AXIS_REF_X2_Slave 		: Tc2_MC2.AXIS_REF;
		AXIS_REF_X3_Slave 		: Tc2_MC2.AXIS_REF;
		                    	
		fbAxis_X1 				: TcAxis_Tc2_MC2;
		fbAxis_Y 				: TcAxis_Tc2_MC2;
		fbAxis_Z 				: TcAxis_Tc2_MC2;
		fbAxis_X2_Slave 		: TcAxis_Tc2_MC2;
		fbAxis_X3_Slave 		: TcAxis_Tc2_MC2;


		Axis_X1 				: itfAxis;
		Axis_Y 					: itfAxis;
		Axis_Z 					: itfAxis;
		Axis_X2_Slave 			: itfAxis;
		Axis_X3_Slave 			: itfAxis;
		                    	
		lastCommandX1 			: itfCommand;
		lastCommandY 			: itfCommand;
		lastCommandZ 			: itfCommand;
		lastCommandX2_slave 	: itfCommand;
		lastCommandX3_slave 	: itfCommand;
		
		targetPosX 				: REAL := 400;
		targetPosY 				: REAL := 600;
		
		ActualPosition_X1 		: REAL;
		ActualPosition_Y 		: REAL;
		ActualPosition_Z 		: REAL;
		ActualPosition_X2_Slave : REAL;
		ActualPosition_X3_Slave : REAL;
		
		ActualVelocity_X1 		: REAL;
		ActualVelocity_Y 		: REAL;
		ActualVelocity_Z 		: REAL;
		ActualVelocity_X2_Slave : REAL;
		ActualVelocity_X3_Slave : REAL;
		
		ActualTorque_X1 		: REAL;
		ActualTorque_Y 			: REAL;
		ActualTorque_Z 			: REAL;
		ActualTorque_X2_Slave 	: REAL;
		ActualTorque_X3_Slave 	: REAL;
					
		Done_X1                 : BOOL;
		Done_Y                  : BOOL;	
		Done_Z                  : BOOL;	
		
	
END_VAR


fbAxis_X1(Axis:=AXIS_REF_X1);
fbAxis_Y(Axis:=AXIS_REF_Y);
fbAxis_Z(Axis:=AXIS_REF_Z);
fbAxis_X2_Slave(Axis:=AXIS_REF_X2_Slave);
fbAxis_X3_Slave(Axis:=AXIS_REF_X3_Slave);

Axis_X1 := fbAxis_X1;
Axis_Y := fbAxis_Y;
Axis_Z := fbAxis_Z;
Axis_X2_Slave := fbAxis_X2_Slave;
Axis_X3_Slave := fbAxis_X3_Slave;

ActualPosition_X1 		:= Axis_X1.ActualPosition;
ActualPosition_Y 		:= Axis_Y.ActualPosition;
ActualPosition_Z 		:= Axis_Z.ActualPosition;
ActualPosition_X2_Slave := Axis_X2_Slave.ActualPosition;
ActualPosition_X3_Slave := Axis_X3_Slave.ActualPosition;

ActualVelocity_X1 		:= Axis_X1.ActualVelocity;
ActualVelocity_Y 		:= Axis_Y.ActualVelocity;
ActualVelocity_Z 		:= Axis_Z.ActualVelocity;
ActualVelocity_X2_Slave := Axis_X2_Slave.ActualVelocity;
ActualVelocity_X3_Slave := Axis_X3_Slave.ActualVelocity;

ActualTorque_X1 		:= Axis_X1.ActualTorque;
ActualTorque_Y 			:= Axis_Y.ActualTorque;
ActualTorque_Z 			:= Axis_Z.ActualTorque;
ActualTorque_X2_Slave 	:= Axis_X2_Slave.ActualTorque;
ActualTorque_X3_Slave 	:= Axis_X3_Slave.ActualTorque;

CASE stateOOP OF
	0: ;
		IF stepOn THEN
			stateOOP := stateOOP + 10;	
		END_IF
	10: 
	// init
		Axis_X1.Power(Enable:=TRUE, EnablePositive:=TRUE, EnableNegative:=TRUE);
		Axis_Y.Power(Enable:=TRUE, EnablePositive:=TRUE, EnableNegative:=TRUE);
		Axis_Z.Power(Enable:=TRUE, EnablePositive:=TRUE, EnableNegative:=TRUE);
		Axis_X2_Slave.Power(Enable:=TRUE, EnablePositive:=TRUE, EnableNegative:=TRUE);
		Axis_X3_Slave.Power(Enable:=TRUE, EnablePositive:=TRUE, EnableNegative:=TRUE);
			
       IF Axis_X1.PowerOn AND Axis_Y.PowerOn AND Axis_Z.PowerOn AND Axis_X2_Slave.PowerOn AND Axis_X3_Slave.PowerOn THEN  	
			IF Axis_X1.Status = Tc2_MC2.MC_AXISSTATE_STANDSTILL AND Axis_Y.Status = Tc2_MC2.MC_AXISSTATE_STANDSTILL AND
				 Axis_Z.Status = Tc2_MC2.MC_AXISSTATE_STANDSTILL AND Axis_X2_Slave.Status = Tc2_MC2.MC_AXISSTATE_STANDSTILL AND Axis_X3_Slave.Status = Tc2_MC2.MC_AXISSTATE_STANDSTILL THEN			
				IF stepOn THEN
					stateOOP := 11;		
					stepOn := FALSE;
				END_IF
			END_IF
		END_IF
	11 : 
	//GearIn
		Axis_X1.GearIn(Slave:= AXIS_REF_X2_Slave, RatioNumerator:= 1,RatioDenominator:= 1, Acceleration:= 0,Deceleration:= 0, Jerk:= 0,BufferMode:= MC_BUFFER_MODE.mcAborting);
		Axis_X1.GearIn(Slave:= AXIS_REF_X3_Slave, RatioNumerator:= 1,RatioDenominator:= 1, Acceleration:= 0,Deceleration:= 0, Jerk:= 0,BufferMode:= MC_BUFFER_MODE.mcAborting);
		stateOOP := 12;						
			
	12:
	// Geared
	    IF Axis_X2_Slave.Geared AND Axis_X3_Slave.Geared THEN			
			stateOOP := 20;
			stepOn := FALSE;		
		END_IF			

	20:
	// start movement in XY
		lastCommandX1 := Axis_X1.MoveAbsolute(Position:=targetPosX, Velocity:=40, Acceleration:=0, Deceleration:=0, Jerk:=0, Direction:=0, BufferMode:=MC_BUFFER_MODE.mcAborting);
		lastCommandY := Axis_Y.MoveAbsolute(Position:=targetPosY, Velocity:=80, Acceleration:=0, Deceleration:=0, Jerk:=0, Direction:=0, BufferMode:=MC_BUFFER_MODE.mcAborting);
			
		Done_X1 S= lastCommandX1.Done;
		Done_Y  S= lastCommandY.Done;
			
		IF Done_X1 AND Done_Y THEN
			stateOOP := stateOOP + 10;					
	  		Done_X1  := FALSE;
			Done_Y   := FALSE;
		END_IF		

	30:
	// wait till movement is finished to 'forkIn'
		Done_Z S= Axis_Z.MoveRelative(Distance:=100, Velocity:=20, Acceleration:=0, Deceleration:=0, Jerk:=0, BufferMode:=MC_BUFFER_MODE.mcAborting).Done;
		IF Done_Z THEN
			stateOOP := stateOOP + 10;
			Done_Z := FALSE;
		END_IF
		
	40:
	// lift pallet if forked in
	    IF NOT Done_X1 THEN
			Done_X1 S= Axis_X1.MoveRelative(Distance:=100, Velocity:=40, Acceleration:=0, Deceleration:=0, Jerk:=0, BufferMode:=MC_BUFFER_MODE.mcAborting).Done;
		END_IF
		IF NOT Done_Y THEN
			Done_Y  S= Axis_Y.MoveRelative(Distance:=100, Velocity:=10, Acceleration:=0, Deceleration:=0, Jerk:=0, BufferMode:=MC_BUFFER_MODE.mcAborting).Done;
		END_IF
		IF Done_X1 AND Done_Y THEN
			stateOOP := stateOOP + 10;
			Done_X1 := FALSE;
			Done_Y  := FALSE;
		END_IF
		
	50:
	// fork out with pallet if forked in is done
		lastCommandZ := Axis_Z.MoveAbsolute(Position:=0, Velocity:=20, Acceleration:=0, Deceleration:=0, Jerk:=0, Direction:=0, BufferMode:=MC_BUFFER_MODE.mcAborting);
		IF lastCommandZ.Done THEN
			stateOOP := stateOOP + 10;
			stepOn := FALSE;
		END_IF

	60:
	// move to delivery if fork out is done
		lastCommandX1 := Axis_X1.MoveAbsolute(Position:=20, Velocity:=40, Acceleration:=0, Deceleration:=0, Jerk:=0, Direction:=0, BufferMode:=MC_BUFFER_MODE.mcAborting);
		lastCommandY := Axis_Y.MoveAbsolute(Position:=20, Velocity:=80, Acceleration:=0, Deceleration:=0, Jerk:=0, Direction:=0, BufferMode:=MC_BUFFER_MODE.mcAborting);

		Done_X1	S= lastCommandX1.Done;
		Done_Y  S= lastCommandY.Done;
			
		IF Done_X1 AND Done_Y THEN			
			stateOOP := stateOOP + 10;
			Done_X1 := FALSE;	
	        Done_Y  := FALSE;
		END_IF

	70:
	// wait till finished	
		Done_X1 S= Axis_X1.MoveAbsolute(Position:=0, Velocity:=20, Acceleration:=0, Deceleration:=0, Jerk:=0, Direction:=0, BufferMode:=MC_BUFFER_MODE.mcAborting).Done;
		Done_Y  S= Axis_Y.MoveAbsolute(Position:=0, Velocity:=20, Acceleration:=0, Deceleration:=0, Jerk:=0, Direction:=0, BufferMode:=MC_BUFFER_MODE.mcAborting).Done;
		IF Done_X1 AND Done_Y THEN
			stateOOP := stateOOP + 10;	
			Done_X1 := FALSE;
			Done_Y  := FALSE;
		END_IF
	80: 
	// ready
	;
END_CASE

END_PROGRAM

// MsTestUnit/FB_Sum
FUNCTION_BLOCK FB_Sum
VAR_INPUT
END_VAR
VAR_OUTPUT
END_VAR
VAR
END_VAR

{attribute 'TcRpcEnable'}
METHOD Sum : INT
VAR_INPUT
	A : INT;
	B : INT;
END_VAR
Sum := A+B;
END_METHOD

END_FUNCTION_BLOCK

// Project Information/F_GetCompany
// This function has been automatically generated from the project information.
{attribute 'signature_flag' := '1073741824'}
{attribute 'TcGenerated'}
{attribute 'no-analysis'}
FUNCTION F_GetCompany : WSTRING
VAR_INPUT
	
END_VAR

F_GetCompany := "TcMotion";

END_FUNCTION

// Project Information/F_GetTitle
// This function has been automatically generated from the project information.
{attribute 'signature_flag' := '1073741824'}
{attribute 'TcGenerated'}
{attribute 'no-analysis'}
FUNCTION F_GetTitle : WSTRING
VAR_INPUT
	
END_VAR

F_GetTitle := "TcMotion_Component";

END_FUNCTION

// Project Information/F_GetVersion
// This function has been automatically generated from the project information.
{attribute 'signature_flag' := '1073741824'}
{attribute 'TcGenerated'}
{attribute 'no-analysis'}
FUNCTION F_GetVersion : ST_LibVersion
VAR_INPUT
	
END_VAR

F_GetVersion.iMajor := 1;
F_GetVersion.iMinor := 0;
F_GetVersion.iBuild := 0;
F_GetVersion.iRevision := 3;
F_GetVersion.sVersion := '1.0.0.3';
F_GetVersion.nFlags := 0;

END_FUNCTION

// TwinCAT Library Template/Part1Definition/Interfaces/itfAxis_Tc2_MC2_Camming
INTERFACE itfAxis_Tc2_MC2_Camming

(*
!!!! It would have to be another library with this new extension for the Axis, because if not in TwinCAT this new license is added:
!!!! TF5050 TC3 NC Camming !!!!!!*)

{warning 'add method implementation '}
METHOD CamIn 			: itfSynchronizedAxisCommand
VAR_INPUT
//	Master				: itfAxis;
	Master				: Tc2_MC2.AXIS_REF;
	Slave				: Tc2_MC2.AXIS_REF;	
	MasterOffset		: REAL;
	SlaveOffset			: REAL;
	MasterScaling		: REAL;
	SlaveScaling		: REAL;
	MasterStartDistance	: REAL;
	MasterSyncPosition	: REAL;
	StartMode			: MC_StartMode;
	MasterValueSource	: MC_Source;
//	CamTable			: itfCamTable;
	CamTableID			: Tc2_MC2_Camming.MC_CAM_ID;
	BufferMode			: MC_BUFFER_MODE;
END_VAR
END_METHOD

END_INTERFACE

// TwinCAT Library Template/Part1Definition/Interfaces/itfAxis_Tc2_MC2_FlyingSaw
INTERFACE itfAxis_Tc2_MC2_FlyingSaw

(*
!!!! It would have to be another library with this new extension for the Axis, because if not in TwinCAT this new license is added:
!!!! TF5055 TC3 NC Flying Saw !!!!!!*)

{warning 'add method implementation '}
METHOD GearInPos 		: itfSynchronizedAxisCommand
VAR_INPUT
//	Master				: itfAxis;
	Master				: Tc2_MC2.AXIS_REF;
	Slave				: Tc2_MC2.AXIS_REF;			
	RatioNumerator		: REAL;
	RatioDenominator	: REAL;
	MasterValueSource	: MC_SOURCE;
	MasterSyncPosition	: REAL;
	SlaveSyncPosition	: REAL;
	SyncMode			: MC_SYNC_MODE;
	MasterStartDistance	: REAL;
	Velocity			: REAL;
	Acceleration		: REAL;
	Deceleration		: REAL;
	Jerk				: REAL;
	BufferMode			: MC_BUFFER_MODE;
END_VAR
END_METHOD

END_INTERFACE

// TwinCAT Library Template/VendorImplementation/TcAxis_DMC_Tc3_Direct_Motion_Control
FUNCTION_BLOCK TcAxis_DMC_Tc3_Direct_Motion_Control IMPLEMENTS itfAxis
VAR_INPUT
	Axis 				: Tc3_Direct_Motion_control.AXIS_REF();
END_VAR
//VAR_OUTPUT
//END_VAR
VAR
END_VAR

END_FUNCTION_BLOCK

// TwinCAT Library Template/VendorImplementation/TcAxis_Tc2_MC2_Camming
FUNCTION_BLOCK TcAxis_Tc2_MC2_Camming EXTENDS TcAxis_Tc2_MC2 IMPLEMENTS itfAxis_Tc2_MC2_Camming
VAR_INPUT
END_VAR
VAR_OUTPUT
END_VAR
VAR
END_VAR

{error 'Agregar implementación de método o eliminar método para utilizar la implementación básica.'}
(*
!!!! It would have to be another library with this new extension for the Axis, because if not in TwinCAT this new license is added:
!!!! TF5050 TC3 NC Camming !!!!!!*)
METHOD CamIn : itfSynchronizedAxisCommand
VAR_INPUT
	(*	Master				: itfAxis;*)
	Master	: Tc2_MC2.AXIS_REF;
	Slave	: Tc2_MC2.AXIS_REF;
	MasterOffset	: REAL;
	SlaveOffset	: REAL;
	MasterScaling	: REAL;
	SlaveScaling	: REAL;
	MasterStartDistance	: REAL;
	MasterSyncPosition	: REAL;
	StartMode	: MC_StartMode;
	MasterValueSource	: MC_Source;
	(*	CamTable			: itfCamTable;*)
	CamTableID	: Tc2_MC2_Camming.MC_CAM_ID;
	BufferMode	: MC_BUFFER_MODE;
END_VAR

VAR
	fbCamIn			 	: Tc2_MC2_Camming.MC_CamIn;	
END_VAR
(*
!!!! It would have to be another library with this new extension for the Axis, because if not in TwinCAT this new license is added:
!!!! TF5050 TC3 NC Camming !!!!!!*)

fbCamIn(
	Master:= Master, 
	Slave:= Slave, 
	Execute:= TRUE, 
	MasterOffset:= MasterOffset, 
	SlaveOffset:= SlaveOffset, 
	MasterScaling:= MasterScaling, 
	SlaveScaling:= SlaveScaling, 
	StartMode:= StartMode, 
	CamTableID:= CamTableID, //CamTable, 
	BufferMode:= , //BufferMode, 
	Options:= , 
	InSync=> , 
	Busy=> , 
	Active=> , 
	CommandAborted=> , 
	Error=> , 
	ErrorID=> );

count_delete  := count_delete + 1;
END_METHOD

END_FUNCTION_BLOCK

// TwinCAT Library Template/VendorImplementation/TcAxis_Tc2_MC2_FlyingSaw
FUNCTION_BLOCK TcAxis_Tc2_MC2_FlyingSaw EXTENDS TcAxis_Tc2_MC2 IMPLEMENTS itfAxis_Tc2_MC2_FlyingSaw
VAR_INPUT
END_VAR
VAR_OUTPUT
END_VAR
VAR
END_VAR

{error 'Agregar implementación de método o eliminar método para utilizar la implementación básica.'}
(*
!!!! It would have to be another library with this new extension for the Axis, because if not in TwinCAT this new license is added:
!!!! TF5055 TC3 NC Flying Saw !!!!!!*)
METHOD GearInPos : itfSynchronizedAxisCommand
VAR_INPUT
	(*	Master				: itfAxis;*)
	Master	: Tc2_MC2.AXIS_REF;
	Slave	: Tc2_MC2.AXIS_REF;
	RatioNumerator	: REAL;
	RatioDenominator	: REAL;
	MasterValueSource	: MC_SOURCE;
	MasterSyncPosition	: REAL;
	SlaveSyncPosition	: REAL;
	SyncMode	: MC_SYNC_MODE;
	MasterStartDistance	: REAL;
	Velocity	: REAL;
	Acceleration	: REAL;
	Deceleration	: REAL;
	Jerk	: REAL;
	BufferMode	: MC_BUFFER_MODE;
END_VAR

VAR
	fbGearInPos			: Tc2_MC2_FlyingSaw.MC_GearInPos;	
END_VAR
(*
!!!! It would have to be another library with this new extension for the Axis, because if not in TwinCAT this new license is added:
!!!! TF5055 TC3 NC Flying Saw !!!!!!*)

fbGearInPos(
	Master:= Master, 
	Slave:= Slave, 
	Execute:= , 
	RatioNumerator:= , 
	RatioDenominator:= , 
	MasterSyncPosition:= , 
	SlaveSyncPosition:= , 
	SyncMode:= , 
	MasterStartDistance:= , 
	Velocity:= , 
	Acceleration:= , 
	Deceleration:= , 
	Jerk:= , 
	BufferMode:= , 
	Options:= , 
	StartSync=> , 
	InSync=> , 
	Busy=> , 
	Active=> , 
	CommandAborted=> , 
	Error=> , 
	ErrorID=> );


count_delete  := count_delete + 1;
END_METHOD

END_FUNCTION_BLOCK

// TwinCAT Library Template/VendorImplementation/TcContinuousAxisCommand
FUNCTION_BLOCK TcContinuousAxisCommand IMPLEMENTS itfContinuousAxisCommand
VAR_INPUT
END_VAR
VAR_OUTPUT
END_VAR
VAR
END_VAR

{warning 'add method implementation '}
METHOD Abort : MC_Error
END_METHOD

{warning 'add property implementation'}
PROPERTY Active : BOOL
GET
END_GET
END_PROPERTY

{warning 'add property implementation'}
PROPERTY Busy : BOOL
GET
END_GET
END_PROPERTY

{warning 'add property implementation'}
PROPERTY Command : MC_COMMAND_REF
GET
END_GET
END_PROPERTY

{warning 'add property implementation'}
PROPERTY CommandAborted : BOOL
GET
END_GET
END_PROPERTY

{warning 'add property implementation'}
PROPERTY Done : BOOL
GET
END_GET
END_PROPERTY

{warning 'add property implementation'}
PROPERTY Error : BOOL
GET
END_GET
END_PROPERTY

{warning 'add property implementation'}
PROPERTY ErrorId : MC_Error
GET
END_GET
END_PROPERTY

{warning 'add property implementation'}
PROPERTY InVelocity : BOOL
GET
END_GET
END_PROPERTY

{warning 'add method implementation '}
METHOD Update 		: MC_Error
VAR_INPUT
	Position		: REAL;
	Velocity		: REAL;
	EndVelocity		: REAL;
	Acceleration	: REAL;
	Deceleration	: REAL;
	Jerk			: REAL;
END_VAR
END_METHOD

{warning 'add method implementation '}
METHOD Wait 		: MC_Error (* This method only makes sense in the IEC 61499 environment*)
VAR_INPUT
	Timeout			: TIME;
	AbortOnTimeout	: BOOL;
END_VAR
END_METHOD

END_FUNCTION_BLOCK

// TwinCAT Library Template/VendorImplementation/TcSynchronizedAxisCommand
FUNCTION_BLOCK TcSynchronizedAxisCommand IMPLEMENTS itfSynchronizedAxisCommand
VAR_INPUT
END_VAR
VAR_OUTPUT
END_VAR
VAR
END_VAR

{warning 'add method implementation '}
METHOD Abort : MC_Error
END_METHOD

{warning 'add property implementation'}
PROPERTY Active : BOOL
GET
END_GET
END_PROPERTY

{warning 'add property implementation'}
PROPERTY Busy : BOOL
GET
END_GET
END_PROPERTY

{warning 'add property implementation'}
PROPERTY Command : MC_COMMAND_REF
GET
END_GET
END_PROPERTY

{warning 'add property implementation'}
PROPERTY CommandAborted : BOOL
GET
END_GET
END_PROPERTY

{warning 'add property implementation'}
PROPERTY Done : BOOL
GET
END_GET
END_PROPERTY

{warning 'add property implementation'}
PROPERTY Error : BOOL
GET
END_GET
END_PROPERTY

{warning 'add property implementation'}
PROPERTY ErrorId : MC_Error
GET
END_GET
END_PROPERTY

{warning 'add property implementation'}
PROPERTY InSync : BOOL
GET
Insync:= Geared;
END_GET
END_PROPERTY

{warning 'add method implementation '}
METHOD Update 		: MC_Error
VAR_INPUT
	Position		: REAL;
	Velocity		: REAL;
	EndVelocity		: REAL;
	Acceleration	: REAL;
	Deceleration	: REAL;
	Jerk			: REAL;
END_VAR
END_METHOD

{warning 'add method implementation '}
METHOD Wait 		: MC_Error (* This method only makes sense in the IEC 61499 environment*)
VAR_INPUT
	Timeout			: TIME;
	AbortOnTimeout	: BOOL;
END_VAR
END_METHOD

END_FUNCTION_BLOCK
